// TwinCAT 3 PLC project RS485_Hausbus_LIB
// Title: RS485_Hausbus_Kernal
// Company: NKAutomation
// Author: N.Kersting
// ProjectVersion: 1.5.0.5
// Description: Der reine RS485 Hausbus Kernal.
// ProgramVersion: 3.1.4026.22
// libraries:
//   Tc2_SerialCom, * (Beckhoff Automation GmbH)
//   Tc2_Standard, * (Beckhoff Automation GmbH)
//   Tc2_System, * (Beckhoff Automation GmbH)
//   Tc3_Module, * (Beckhoff Automation GmbH)
// project tree:
//   DUTs/HausBus/BusTaster/ ST_BusTaster6F_Cnt.TcDUT, ST_BusTaster6F_Input.TcDUT, ST_BusTaster6F_Output.TcDUT
//   DUTs/HausBus/CMD/ E_EnumHBCmdRX.TcDUT, E_EnumHBCmdTX.TcDUT, E_EnumHBUnitTX.TcDUT
//   DUTs/HausBus/CYD/ ST_BusCYD6F_Input.TcDUT
//   DUTs/HausBus/Dimmer/ ST_6FDimm.TcDUT, ST_BusDimmer6F_Input.TcDUT, ST_BusDimmer6F_Output.TcDUT
//   DUTs/HausBus/ E_EnumHBDeviceOPMode.TcDUT, E_EnumHBDeviceType.TcDUT, ST_HausBus_Ident.TcDUT
//   DUTs/HausBus/RelaisModul/ ST_16Relais.TcDUT, ST_BusRelais16F_Cnt.TcDUT, ST_BusRelais16F_Input.TcDUT, ST_BusRelais16F_Output.TcDUT
//   DUTs/HausBus/Service/ ST_FiFoMaster_State.TcDUT, ST_RS485ComDeviceStatus.TcDUT, ST_RS485Startup_State.TcDUT
//   DUTs/HausBus/TempSensor/ ST_BusTempSensor4F_Input.TcDUT, ST_BusTempSensor4F_Output.TcDUT
//   GVLs/RS485_HausBus/ GVL_HausBus_ASCII_CONSTANT.TcGVL, GVL_HausBus_CONSTANT.TcGVL, GVL_HausBus_Functions.TcGVL, GVL_HausBus_States.TcGVL, GVL_Times.TcGVL
//   / PlcTask.TcTTO
//   POUs/Hilfsbausteine/ fb_timeDiffLite_libversion.TcPOU
//   POUs/ MAIN.TcPOU
//   POUs/RS485_Hausbus_FB/00_CMD/ fb_RS485HB_StringBuilder.TcPOU, F_RS485HB_TO_ASCII.TcPOU, F_RS485HB_TO_ASCII_RX.TcPOU, F_RS485HB_TO_ASCII_RX_PING.TcPOU
//   POUs/RS485_Hausbus_FB/00_Events/ fb_BusBrsEvent.TcPOU, fb_BusDimmEvent.TcPOU, fb_BusPingEvent.TcPOU (not stored), fb_BusRhdEvent.TcPOU, fb_BusTasterAdvancedEvent_4F.TcPOU, fb_BusTasterAdvancedEvent_6F.TcPOU, fb_BusTasterAdvancedEvent_8F.TcPOU, fb_BusTempEvent.TcPOU
//   POUs/RS485_Hausbus_FB/00_RS485 COM/FB/ fb_FilterArray.TcPOU
//   POUs/RS485_Hausbus_FB/00_RS485 COM/ fb_RS485IdScan.TcPOU
//   POUs/RS485_Hausbus_FB/00_RS485 COM/OLD/ fb_RS485Ping.TcPOU
//   POUs/RS485_Hausbus_FB/00_RS485 COM/RS485_Master/ fb_RS485FiFoMaster.TcPOU, fb_RS485Logger.TcPOU, fb_RS485Startup.TcPOU
//   POUs/RS485_Hausbus_FB/01_BusTaster/ fb_TasterBus6F.TcPOU
//   POUs/RS485_Hausbus_FB/01_CYD/ fb_BusTasterEvent.TcPOU, fb_CYDBus6F.TcPOU, fb_StringConvCYDService.TcPOU, fb_StringConvCYDWeb.TcPOU, fb_StringConvCYDWifi.TcPOU, fb_StringConvTB6F.TcPOU
//   POUs/RS485_Hausbus_FB/01_Dimmer/ fb_DimmerBus6F.TcPOU
//   POUs/RS485_Hausbus_FB/01_RelaisModul/ fb_RelaisBus16F.TcPOU
//   POUs/RS485_Hausbus_FB/01_TempSensor/ fb_TempBus4F.TcPOU
//   POUs/RS485_Hausbus_FB/02_UniBaustein/ fb_RS485PingCheck.TcPOU, fb_UniHBComOperator.TcPOU
//   Project Information/ F_GetCompany.TcPOU, F_GetTitle.TcPOU, F_GetVersion.TcPOU
//   Version/ Global_Version.TcGVL

CONFIGURATION RS485_Hausbus_LIB
    RESOURCE PLC ON TwinCAT3
        TASK PlcTask(INTERVAL := T#10ms, PRIORITY := 20);
        PROGRAM MAIN WITH PlcTask : MAIN;
    END_RESOURCE
END_CONFIGURATION

// ---- DUTs/HausBus/BusTaster/ST_BusTaster6F_Cnt.TcDUT
TYPE ST_BusTaster6F_Cnt :
STRUCT
	dwCntButtons    :ARRAY[1..6] OF DWORD;
END_STRUCT
END_TYPE

// ---- DUTs/HausBus/BusTaster/ST_BusTaster6F_Input.TcDUT
TYPE ST_BusTaster6F_Input :
STRUCT
	diID		:DINT;							(* Device ID ( Steht auf dem Aufkleber und wird zur Identifizierung im BUS benötigt)*)
	sName		:STRING;						(* Name des Tasters (zb- Wohnzimmer1 *)
	iLED      	:ARRAY[1..6] OF INT;     	  	(* gewünschter LED-Zustand (TRUE = 100 %)*)
	iLEDExt    	:ARRAY[1..6] OF INT;     	  	(* gewünschter LED-Zustand (TRUE = 100 %)*)
	iLEDBg		:INT;							(* gewünschte Hintergrundbeleuchtung *)
	bReset		:BOOL;							(* Reset des Tasters (Hardware) *)
	bExecute	:BOOL;							(* Aktivierung des Tasters *)
	bExtOutLED	:BOOL;							(* Verwendet die  Extra Ausgänge für LEDs / Mehr Busaulastung!  *)
	bExtInputs	:BOOL := FALSE;					(* Aktiviert die Externen Inputs *)
END_STRUCT
END_TYPE

// ---- DUTs/HausBus/BusTaster/ST_BusTaster6F_Output.TcDUT
TYPE ST_BusTaster6F_Output :
STRUCT
	bButtons    :ARRAY[1..6] OF BOOL;       (*aktueller Tasterstatus (TRUE = gedrückt)*)
	bButtonsExt :ARRAY[1..6] OF BOOL;       (*aktueller Tasterstatus (TRUE = gedrückt)*)
	
	lrTemp		:LREAL;						(* Temperatur Sensor	*)
	lrRhd		:LREAL;						(* Luftfeuchtigkeit Sensor	*)
	lrBrs		:LREAL;						(* Helligkeit Sensor *)
	
	bCOM			:BOOL;					(*Zeigt die Kommunikation an *)
	bStartupDone	:BOOL;
	
	iState			:BOOL;
	sState			:STRING;
	bError			:BOOL;
	
	tLastUpdateTemp	:TIME;					(* Zeit- Letztes Update Temperatur *)
	tLastUpdateRhd	:TIME;					(* Zeit- Letztes Update Luftfeuchte *)
	tLastUpdateBrs	:TIME;					(* Zeit- Letztes Update Helligkeit *)
	
	sLastUpdateTemp	:STRING(12);			(* Zeit- Letztes Update Temperatur Uhrzeit *)
	sLastUpdateRhd	:STRING(12);			(* Zeit- Letztes Update Luftfeuchte Uhrzeit*)
	sLastUpdateBrs	:STRING(12);			(* Zeit- Letztes Update Helligkeit Uhrzeit*)
	
	dwChanges		:DWORD;					(* Änderungszähler für Startups *)
END_STRUCT
END_TYPE

// ---- DUTs/HausBus/CMD/E_EnumHBCmdRX.TcDUT
{attribute 'qualified_only'}
{attribute 'strict'}
{attribute 'to_string'}
TYPE E_EnumHBCmdRX :
(	
	E_HB_CMD_STATUS := 0,		(* STATUS*)
	E_HB_CMD_rSTATUS := 10,		(* rSTATUS*)
	E_HB_CMD_rCONFIG := 11		(* rCONFIG*)
);
END_TYPE

// ---- DUTs/HausBus/CMD/E_EnumHBCmdTX.TcDUT
{attribute 'qualified_only'}
{attribute 'strict'}
{attribute 'to_string'}
TYPE E_EnumHBCmdTX :
(	
	E_HB_CMD_RESET := 0,	(* RESET*)
	E_HB_CMD_gSTATUS := 100,	(* gSTATUS*)
	E_HB_CMD_gCONFIG := 101,	(* gCONFIG*)
	E_HB_CMD_SET_CFG := 200,	(* SET_CFG*)
	E_HB_CMD_ON := 201,	(* ON*)
	E_HB_CMD_OFF := 202,	(* OFF*)
	E_HB_CMD_SET_MBR := 203,	(* SET_MBR*)
	E_HB_CMD_ON_NP := 204,	(* ON _OHNE Parameter *)
	E_HB_CMD_ON_OFF := 205	(* ON _OFF_ nur über Parameter *)
);
END_TYPE

// ---- DUTs/HausBus/CMD/E_EnumHBUnitTX.TcDUT
{attribute 'qualified_only'}
{attribute 'strict'}
{attribute 'to_string'}
TYPE E_EnumHBUnitTX :
(	
	E_HB_UNIT_SYS := 0,		(* SYS*)
	E_HB_UNIT_BTN := 10,	(* BTN*)
	E_HB_UNIT_OUT := 11,	(* OUT*)
	E_HB_UNIT_LED := 12,	(* LED*)
	E_HB_UNIT_TMP := 13,	(* TMP*)
	E_HB_UNIT_RHD := 14,	(* RHD*)
	E_HB_UNIT_BRS := 15,	(* BRS*)
	E_HB_UNIT_DIM := 16,	(* DIM*)
	E_HB_UNIT_LBN := 17		(* LBN*)
);
END_TYPE

// ---- DUTs/HausBus/CYD/ST_BusCYD6F_Input.TcDUT
TYPE ST_BusCYD6F_Input :
STRUCT
	diID			:DINT;							(* Device ID ( Steht auf dem Aufkleber und wird zur Identifizierung im BUS benötigt)*)
	sName			:STRING;						(* Name des Tasters (zb- Wohnzimmer1 *)
	iLED      		:ARRAY[1..6] OF INT;     	  	(* gewünschter LED-Zustand (TRUE = 100 %)*)
	iLEDExt   	 	:ARRAY[1..6] OF INT;     	  	(* gewünschter LED-Zustand (TRUE = 100 %)*)
	iLEDBg			:INT;							(* gewünschte Hintergrundbeleuchtung *)
	
	
	bReset			:BOOL;							(* Reset des Tasters (Hardware) *)
	bExecute		:BOOL;							(* Aktivierung des Tasters *)
	bExtOutLED		:BOOL;							(* Verwendet die  Extra Ausgänge für LEDs / Mehr Busaulastung!  *)
	
	bServiceMode	:BOOL;
	bService		:BOOL;
	bWifi			:BOOL;
	bWebServer		:BOOL;
END_STRUCT
END_TYPE

// ---- DUTs/HausBus/Dimmer/ST_6FDimm.TcDUT
TYPE ST_6FDimm :
STRUCT
	sLocation			:STRING(28);	
	iDimm	 : ARRAY[1..6] OF INT;
END_STRUCT
END_TYPE

// ---- DUTs/HausBus/Dimmer/ST_BusDimmer6F_Input.TcDUT
TYPE ST_BusDimmer6F_Input :
STRUCT
	diID		:DINT;							(* Device ID ( Steht auf dem Aufkleber und wird zur Identifizierung im BUS benötigt)*)
	sName		:STRING;						(* Name des Tasters (zb- Wohnzimmer1 *)
	iLED      	:ARRAY[1..6] OF INT;     	  	(* gewünschter LED-Zustand (TRUE = 100 %)*)
	iDimmspeed	:INT :=10;						(* Dimmerrampe für alle Kanäle  *)
	bWriteCfg	:BOOL := FALSE;					(* Config write ausführen  *)
	bReset		:BOOL;							(* Reset des Tasters (Hardware) *)
	bExecute	:BOOL;							(* Aktivierung des Tasters *)
	bExtInputs	:BOOL := FALSE;					(* Aktiviert die Externen Inputs *)
END_STRUCT
END_TYPE

// ---- DUTs/HausBus/Dimmer/ST_BusDimmer6F_Output.TcDUT
TYPE ST_BusDimmer6F_Output :
STRUCT
	bInputs		    :ARRAY[1..4] OF BOOL;       (*aktueller Input Status (TRUE = gedrückt)*)
	bCOM			:BOOL;						(*Zeigt die Kommunikation an *)
	bStartupDone	:BOOL;
	
	iState			:BOOL;
	sState			:STRING;
	bError			:BOOL;
	dwChanges		:DWORD;					(* Änderungszähler für Startups *)
END_STRUCT
END_TYPE

// ---- DUTs/HausBus/E_EnumHBDeviceOPMode.TcDUT

TYPE E_EnumHBDeviceOPMode :
(
	E_HB_Device_Init,
	E_HB_Device_CheckID,
	E_HB_Device_EventStartup,
	E_HB_Device_Reset,
	E_HB_Device_WaitCom,
	E_HB_Device_Startup,
	E_HB_Device_OP
);
END_TYPE

// ---- DUTs/HausBus/E_EnumHBDeviceType.TcDUT
TYPE E_EnumHBDeviceType :
(
	E_HB_Device_NV ,
	E_HB_Device_6FTaster,
	E_HB_Device_16FRelais,
	E_HB_Device_6FDimmer,
	E_HB_Device_CYD_1
	
);
END_TYPE

// ---- DUTs/HausBus/RelaisModul/ST_16Relais.TcDUT
TYPE ST_16Relais :
STRUCT
	sLocation			:STRING(28);	
	bOut	 : ARRAY[1..16] OF BOOL;
END_STRUCT
END_TYPE

// ---- DUTs/HausBus/RelaisModul/ST_BusRelais16F_Cnt.TcDUT
TYPE ST_BusRelais16F_Cnt :
STRUCT
	dwCntRelais    :ARRAY[1..16] OF DWORD;
END_STRUCT
END_TYPE

// ---- DUTs/HausBus/RelaisModul/ST_BusRelais16F_Input.TcDUT
TYPE ST_BusRelais16F_Input :
STRUCT
	diID		:DINT;							(* Device ID ( Steht auf dem Aufkleber und wird zur Identifizierung im BUS benötigt)*)
	sName		:STRING;						(* Name des Tasters (zb- Wohnzimmer1 *)
	bOut     	:ARRAY[1..16] OF BOOL;     	  	(* gewünschter Zustand (TRUE = An%)*)
	bReset		:BOOL;							(* Reset des Tasters (Hardware) *)
	bExecute	:BOOL;							(* Aktivierung des Tasters *)
	bExtInputs	:BOOL := FALSE;					(* Aktiviert die Externen Inputs *)
END_STRUCT
END_TYPE

// ---- DUTs/HausBus/RelaisModul/ST_BusRelais16F_Output.TcDUT
TYPE ST_BusRelais16F_Output :
STRUCT
	bInputs		    :ARRAY[1..8] OF BOOL;       (*aktueller Tasterstatus (TRUE = gedrückt)*)
	bCOM			:BOOL;					(*Zeigt die Kommunikation an *)
	bStartupDone	:BOOL;
	
	iState			:BOOL;
	sState			:STRING;
	bError			:BOOL;
	dwChanges		:DWORD;					(* Änderungszähler für Startups *)
END_STRUCT
END_TYPE

// ---- DUTs/HausBus/Service/ST_FiFoMaster_State.TcDUT
TYPE ST_FiFoMaster_State :
STRUCT
	sReceiveString			:STRING(255);		
	lrBusAuslastung			:LREAL;
	bBusy					:BOOL;
	bDone					:BOOL;
	bError					:BOOL;
	iFiFoCount				:INT;
	iFiFoRow				:INT;
	sSendString				:STRING(255);
	sState					:STRING;
	
END_STRUCT
END_TYPE

// ---- DUTs/HausBus/Service/ST_RS485ComDeviceStatus.TcDUT
TYPE ST_RS485ComDeviceStatus :
STRUCT
	diID			:DINT;			
	sState			:STRING;
	bCOM			:BOOL;					(*Zeigt die Kommunikation an *)
	bStartupDone	:BOOL;
	bError			:BOOL;
	
	(* Vorbehalt für Taster *)
	lrTemp			:LREAL;						(* Temperatur Sensor	*)
	lrRhd			:LREAL;						(* Luftfeuchtigkeit Sensor	*)
	lrBrs			:LREAL;						(* Helligkeit Sensor *)
		
	dwChanges		:DWORD;				
END_STRUCT
END_TYPE

// ---- DUTs/HausBus/Service/ST_RS485Startup_State.TcDUT
TYPE ST_RS485Startup_State :
STRUCT
	bBusOk					:BOOL;
	bStartupError			:BOOL;
	sStartupState			:STRING;
	bStartupDone			:BOOL;
END_STRUCT
END_TYPE

// ---- DUTs/HausBus/ST_HausBus_Ident.TcDUT
TYPE ST_HausBus_Ident :
STRUCT
	diID			:DINT;							(* Device ID ( Steht auf dem Aufkleber und wird zur Identifizierung im BUS benötigt)*)
	sName			:STRING;						(* Name des Tasters (zb- Wohnzimmer1 *)	
	sPingIdent		:STRING :='TMP.1.gSTATUS'; 		(* Ping Identifiaktions String, wird bim Pingen gesendet  (Bei Taster = TMP.1.gSTATUS / Relais = OUT.210.rSTATUS / CYD= noch nicht definiert*)
	bUseExtInputs	:BOOL := FALSE;					(* Aktiviert die Externen Inputs *)
END_STRUCT
END_TYPE

// ---- DUTs/HausBus/TempSensor/ST_BusTempSensor4F_Input.TcDUT
TYPE ST_BusTempSensor4F_Input :
STRUCT
	diID		:DINT;							(* Device ID ( Steht auf dem Aufkleber und wird zur Identifizierung im BUS benötigt)*)
	sName		:STRING;						(* Name des Tasters (zb- Wohnzimmer1 *)
	bReset		:BOOL;							(* Reset des ESP32 (Hardware) *)
	bExecute	:BOOL;							(* Aktivierung des Sensors *)
	
	iAnzTempSens :INT := 4;						(* Anzahl der Tempsensoren *)
	bExtInputs	:BOOL := FALSE;					(* Aktiviert die Externen Inputs *)
	
	bWifi			:BOOL;
END_STRUCT
END_TYPE

// ---- DUTs/HausBus/TempSensor/ST_BusTempSensor4F_Output.TcDUT
TYPE ST_BusTempSensor4F_Output :
STRUCT	
	lrTemp			:ARRAY[1..4] OF LREAL;					(* Temperatur Sensor	*)
	
	bCOM			:BOOL;					(*Zeigt die Kommunikation an *)
	bStartupDone	:BOOL;
	
	iState			:BOOL;
	sState			:STRING;
	bError			:BOOL;
	
	tLastUpdateTemp	:ARRAY[1..4] OF TIME;					(* Zeit- Letztes Update Temperatur *)
	
	sLastUpdateTemp	:ARRAY[1..4] OF STRING(12);			(* Zeit- Letztes Update Temperatur Uhrzeit *)
	
	dwChanges		:DWORD;					(* Änderungszähler für Startups *)
END_STRUCT
END_TYPE

// ---- GVLs/RS485_HausBus/GVL_HausBus_ASCII_CONSTANT.TcGVL
{attribute 'qualified_only'}
VAR_GLOBAL CONSTANT
(*==================================================================*)
(* Bibliothek aller ASCII Befehle für alle HAUS-BUS Komponenten *)
(*==================================================================*)

HB_UNIT_SYS : STRING(3) := 'SYS';	(* <SYS>	System *)
HB_UNIT_BRS : STRING(3) := 'BRS';	(* <BRS>	Helligkeit *)
HB_UNIT_BTN : STRING(3) := 'BTN';	(* <BTN>	Button *)
HB_UNIT_DIM : STRING(3) := 'DIM';	(* <DIM>	Dimmer *)
HB_UNIT_LED : STRING(3) := 'LED';	(* <LED>	LED/ Ausgang Taster *)
HB_UNIT_OUT : STRING(3) := 'OUT';	(* <OUT>	Ausgang z.B. Relaismodule  *)
HB_UNIT_RHD : STRING(3) := 'RHD';	(* <RHD>	Luftfeuchtigkeit  *)
HB_UNIT_TMP : STRING(3) := 'TMP';	(* <TMP>	Temperatur  *)
HB_UNIT_LBN : STRING(3) := 'LBN';	(* <LBN>	Hintergrundbeleuchtung (Von Taster) *)

HB_CMD_RESET 	: STRING(7) := 'RESET';		(* <RESET>		Reset des Devices anfordern *)
HB_CMD_gCONFIG 	: STRING(7) := 'gCONFIG';	(* <gCONFIG> 	Config abfragen *)
HB_CMD_gSTATUS 	: STRING(7) := 'gSTATUS';	(* <gSTATUS> 	STATUS abfragen *)
HB_CMD_OFF	 	: STRING(7) := 'OFF';		(* <OFF>		Off Befehl mit Steuerung über Parameter *)
HB_CMD_ON	 	: STRING(7) := 'ON';		(* <ON>			ON Befehl mit Steuerung über Parameter *)
HB_CMD_SET_CFG 	: STRING(7) := 'SET_CFG';	(* <SET_CFG>	Setze Config  *)
HB_CMD_SET_MBR 	: STRING(7) := 'SET_MBR';	(* <SET_MBR>	Setze Hintergrundhelligkeit *)
HB_CMD_ON_NP 	: STRING(7) := 'ON';		(* <ON>			SONDERFUNKTION! Besitzt keine Parameter!  *)
HB_CMD_ON_OFF 	: STRING(7) := '';			(* <ON>			SONDERFUNKTION! Wird über den Parametereingang gesteuert! Wenn P=1 dann 'ON'  wenn P=2 dann 'OFF' *)

HB_RX_rCONFIG	: STRING(7) := 'rCONFIG';	(* <rCONFIG>	Empfang von Config *)
HB_RX_STATUS	: STRING(7) := 'STATUS';	(* <STATUS>		Empfang von Statusnachricht *)
HB_RX_rSTATUS	: STRING(7) := 'rSTATUS';	(* <rSTATUS>	Empfang von Statusantwort *)
END_VAR

// ---- GVLs/RS485_HausBus/GVL_HausBus_CONSTANT.TcGVL
{attribute 'Tc2GvlVarNames'}
VAR_GLOBAL CONSTANT
	(*FiFo*)
	cMaxRowCMDFiFo			:INT := 50; (* Anzahl Maximal mögliche FiFo Zeilen *)
	cMaxScanIDs				:INT := 50;
END_VAR

// ---- GVLs/RS485_HausBus/GVL_HausBus_Functions.TcGVL
{attribute 'Tc2GvlVarNames'}
VAR_GLOBAL
(*================================================================================================================================*)		
(* Changecounter aller Teilnehmer zurücksetzen *)		
(*================================================================================================================================*)	
	bResetChangesCounter_All			:BOOL := FALSE;
END_VAR

// ---- GVLs/RS485_HausBus/GVL_HausBus_States.TcGVL
{attribute 'Tc2GvlVarNames'}
VAR_GLOBAL
	bGlobalPingActive	:BOOL;
END_VAR

// ---- GVLs/RS485_HausBus/GVL_Times.TcGVL
{attribute 'Tc2GvlVarNames'}
VAR_GLOBAL
	
	sGlobClock_SMH					:STRING(12);
END_VAR

// ---- Version/Global_Version.TcGVL
{attribute 'TcGenerated'}
{attribute 'no-analysis'}
{attribute 'linkalways'}
// This function has been automatically generated from the project information.
VAR_GLOBAL CONSTANT
	{attribute 'const_non_replaced'}
	stLibVersion_RS485_Hausbus_Kernal : ST_LibVersion := (iMajor := 1, iMinor := 5, iBuild := 0, iRevision := 5, nFlags := 1, sVersion := '1.5.0.5');
END_VAR

// ---- POUs/MAIN.TcPOU
PROGRAM MAIN
VAR
END_VAR

END_PROGRAM

// ---- POUs/Hilfsbausteine/fb_timeDiffLite_libversion.TcPOU
(*======================================================================================================================================*)
(*fb_timeDiffLite:	Neuer einfacherer Baustein, welcher nur über Start funktioniert *)
(*
Date          	| Version    	| created under        	| Author          	| Remark *)
(*======================================================================================================================================*)
(*03/09/2025   	| 1.00      	| TC3		  			| N.Kersting       | first release *)
(*======================================================================================================================================*)
FUNCTION_BLOCK fb_timeDiffLite_libversion
VAR_INPUT
	I_bStart	:BOOL;
	I_bReset	:BOOL;
END_VAR
VAR_OUTPUT
	Q_tDiffTime	:TIME;
END_VAR
VAR
	tStart	:TIME;
	tStop	:TIME;

	rTrigStart:	R_TRIG;
	rTrigStop:	R_TRIG;
	bMem: BOOL;
END_VAR

rTrigStart(CLK:=I_bStart);

IF	I_bReset	
THEN	
	bMem := FALSE;
	tStart:= T#0S;
	tStop:=T#0S;
ELSE
	
	IF	rTrigStart.Q	
		AND bMem
	THEN	
		bMem := FALSE; 
		tStart:= TIME();
		Q_tDiffTime:=	tStart-tStop;
	END_IF

	IF	rTrigStart.Q
		AND NOT bMem	
	THEN	
		bMem := TRUE;
		tStop:=	TIME();
	END_IF
END_IF

END_FUNCTION_BLOCK

// ---- POUs/RS485_Hausbus_FB/00_CMD/fb_RS485HB_StringBuilder.TcPOU
(*======================================================================================================================================*)
(*//=============================================================================\\
||  _   _ _  __  _         _                        _   _                      ||
|| | \ | | |/ / / \  _   _| |_ ___  _ __ ___   __ _| |_(_) ___  _ __         ||
|| |  \| | ' / / _ \| | | | __/ _ \| '_ ` _ \ / _` | __| |/ _ \| '_ \        ||
|| | |\  | . \/ ___ \ |_| | || (_) | | | | | | (_| | |_| | (_) | | | |       ||
|| |_| \_|_|\_\_/  \_\__,_|\__\___/|_| |_| |_|\__,_|\__|_|\___/|_| |_|       ||
||                                                                             ||
\\=============================================================================//
fb_RS485HB_StringBuilder:	Funktionsbaustein zum zusammenbauen komplexer Strings für Hausbus RS485 Ascii Telegramme		*)
(*
Date          	| Version    	| created under        	| Author          	| Remark *)
(*====================================================================================================================================================*)
(*22/01/2026   	| 1.00      	| TC3		  			| N.Kersting        | first release *)
(*22/01/2026   	| 1.01      	| TC3		  			| N.Kersting        | Erweiterung Array auf 8 Index *)
(*====================================================================================================================================================*)
FUNCTION_BLOCK fb_RS485HB_StringBuilder
VAR_INPUT
	I_bExecute			:BOOL := FALSE;
	I_diID				:DINT;				(* Device ID ( Steht auf dem Aufkleber und wird zur Identifizierung im BUS benötigt)*)
	I_iInstID			:INT;				(* Instanz ID *)
	I_EnumHBUnitTX		:E_EnumHBUnitTX;	(* Unit *)
	I_EnumHBCmdTX		:E_EnumHBCmdTX;		(* Command *)
	I_iCnt				:INT;				(* Anzahl der zusammengefügten Befehle *)
	I_iP1				:ARRAY[1..8] OF INT;				(* Parameter 1 *)
	I_iP2				:ARRAY[1..8] OF INT;				(* Parameter 2 *)
	I_iP3				:ARRAY[1..8] OF INT;				(* Parameter 3 *)
	I_iP4				:ARRAY[1..8] OF INT;				(* Parameter 4 *)
END_VAR
VAR_OUTPUT	
	Q_sOut				:STRING(255);							(* Fertiger Ausgabestring*)	
	Q_bDone				:BOOL;
	Q_bError			:BOOL;
END_VAR
VAR
	IDX 				:INT;
	Trig				:r_trig;
	nLength				:INT;
END_VAR

Trig(CLK:=I_bExecute);

IF Trig.Q
	AND I_bExecute
THEN
	IF I_diID <> 0
	THEN
		IF I_iInstID <> 0
		THEN
			IF I_iCnt <>0
				AND I_iCnt <=8
			THEN
				Q_bError := FALSE;
				
				CASE I_iCnt OF
				(*===========================*)
				0: 	IDX := 0;
					Q_sOut :='';
					
					Q_bDone := TRUE;
					RETURN;
					
				(*===========================*)
				1: 	IDX := 1;
					Q_sOut 	:=		F_RS485HB_TO_ASCII(I_diID,I_iInstID,I_EnumHBUnitTX,I_EnumHBCmdTX,I_iP1[IDX],I_iP2[IDX],I_iP3[IDX],I_iP4[IDX]);
					
					Q_bDone := TRUE;
					
				(*===========================*)
				2: 	IDX := 1;
					Q_sOut 	:=		F_RS485HB_TO_ASCII(I_diID,I_iInstID,I_EnumHBUnitTX,I_EnumHBCmdTX,I_iP1[IDX],I_iP2[IDX],I_iP3[IDX],I_iP4[IDX]);
					IDX := 2;
					Q_sOut 	:=		CONCAT(Q_sOut,F_RS485HB_TO_ASCII(I_diID,I_iInstID+IDX-1,I_EnumHBUnitTX,I_EnumHBCmdTX,I_iP1[IDX],I_iP2[IDX],I_iP3[IDX],I_iP4[IDX]));
					
					Q_bDone := TRUE;
					
				(*===========================*)
				3: 	IDX := 1;
					Q_sOut 	:=		F_RS485HB_TO_ASCII(I_diID,I_iInstID,I_EnumHBUnitTX,I_EnumHBCmdTX,I_iP1[IDX],I_iP2[IDX],I_iP3[IDX],I_iP4[IDX]);
					IDX := 2;
					Q_sOut 	:=		CONCAT(Q_sOut,F_RS485HB_TO_ASCII(I_diID,I_iInstID+IDX-1,I_EnumHBUnitTX,I_EnumHBCmdTX,I_iP1[IDX],I_iP2[IDX],I_iP3[IDX],I_iP4[IDX]));
					IDX := 3;
					Q_sOut 	:=		CONCAT(Q_sOut,F_RS485HB_TO_ASCII(I_diID,I_iInstID+IDX-1,I_EnumHBUnitTX,I_EnumHBCmdTX,I_iP1[IDX],I_iP2[IDX],I_iP3[IDX],I_iP4[IDX]));
					
					Q_bDone := TRUE;
					
				(*===========================*)
				4: 	IDX := 1;
					Q_sOut 	:=		F_RS485HB_TO_ASCII(I_diID,I_iInstID,I_EnumHBUnitTX,I_EnumHBCmdTX,I_iP1[IDX],I_iP2[IDX],I_iP3[IDX],I_iP4[IDX]);
					IDX := 2;
					Q_sOut 	:=		CONCAT(Q_sOut,F_RS485HB_TO_ASCII(I_diID,I_iInstID+IDX-1,I_EnumHBUnitTX,I_EnumHBCmdTX,I_iP1[IDX],I_iP2[IDX],I_iP3[IDX],I_iP4[IDX]));
					IDX := 3;
					Q_sOut 	:=		CONCAT(Q_sOut,F_RS485HB_TO_ASCII(I_diID,I_iInstID+IDX-1,I_EnumHBUnitTX,I_EnumHBCmdTX,I_iP1[IDX],I_iP2[IDX],I_iP3[IDX],I_iP4[IDX]));
					IDX := 4;
					Q_sOut 	:=		CONCAT(Q_sOut,F_RS485HB_TO_ASCII(I_diID,I_iInstID+IDX-1,I_EnumHBUnitTX,I_EnumHBCmdTX,I_iP1[IDX],I_iP2[IDX],I_iP3[IDX],I_iP4[IDX]));
					
					Q_bDone := TRUE;
					
				(*===========================*)
				5: 	IDX := 1;
					Q_sOut 	:=		F_RS485HB_TO_ASCII(I_diID,I_iInstID,I_EnumHBUnitTX,I_EnumHBCmdTX,I_iP1[IDX],I_iP2[IDX],I_iP3[IDX],I_iP4[IDX]);
					IDX := 2;
					Q_sOut 	:=		CONCAT(Q_sOut,F_RS485HB_TO_ASCII(I_diID,I_iInstID+IDX-1,I_EnumHBUnitTX,I_EnumHBCmdTX,I_iP1[IDX],I_iP2[IDX],I_iP3[IDX],I_iP4[IDX]));
					IDX := 3;
					Q_sOut 	:=		CONCAT(Q_sOut,F_RS485HB_TO_ASCII(I_diID,I_iInstID+IDX-1,I_EnumHBUnitTX,I_EnumHBCmdTX,I_iP1[IDX],I_iP2[IDX],I_iP3[IDX],I_iP4[IDX]));
					IDX := 4;
					Q_sOut 	:=		CONCAT(Q_sOut,F_RS485HB_TO_ASCII(I_diID,I_iInstID+IDX-1,I_EnumHBUnitTX,I_EnumHBCmdTX,I_iP1[IDX],I_iP2[IDX],I_iP3[IDX],I_iP4[IDX]));
					IDX := 5;
					Q_sOut 	:=		CONCAT(Q_sOut,F_RS485HB_TO_ASCII(I_diID,I_iInstID+IDX-1,I_EnumHBUnitTX,I_EnumHBCmdTX,I_iP1[IDX],I_iP2[IDX],I_iP3[IDX],I_iP4[IDX]));
					
					Q_bDone := TRUE;
					
				(*===========================*)
				6: 	IDX := 1;
					Q_sOut 	:=		F_RS485HB_TO_ASCII(I_diID,I_iInstID,I_EnumHBUnitTX,I_EnumHBCmdTX,I_iP1[IDX],I_iP2[IDX],I_iP3[IDX],I_iP4[IDX]);
					IDX := 2;
					Q_sOut 	:=		CONCAT(Q_sOut,F_RS485HB_TO_ASCII(I_diID,I_iInstID+IDX-1,I_EnumHBUnitTX,I_EnumHBCmdTX,I_iP1[IDX],I_iP2[IDX],I_iP3[IDX],I_iP4[IDX]));
					IDX := 3;
					Q_sOut 	:=		CONCAT(Q_sOut,F_RS485HB_TO_ASCII(I_diID,I_iInstID+IDX-1,I_EnumHBUnitTX,I_EnumHBCmdTX,I_iP1[IDX],I_iP2[IDX],I_iP3[IDX],I_iP4[IDX]));
					IDX := 4;
					Q_sOut 	:=		CONCAT(Q_sOut,F_RS485HB_TO_ASCII(I_diID,I_iInstID+IDX-1,I_EnumHBUnitTX,I_EnumHBCmdTX,I_iP1[IDX],I_iP2[IDX],I_iP3[IDX],I_iP4[IDX]));
					IDX := 5;
					Q_sOut 	:=		CONCAT(Q_sOut,F_RS485HB_TO_ASCII(I_diID,I_iInstID+IDX-1,I_EnumHBUnitTX,I_EnumHBCmdTX,I_iP1[IDX],I_iP2[IDX],I_iP3[IDX],I_iP4[IDX]));
					IDX := 6;
					Q_sOut 	:=		CONCAT(Q_sOut,F_RS485HB_TO_ASCII(I_diID,I_iInstID+IDX-1,I_EnumHBUnitTX,I_EnumHBCmdTX,I_iP1[IDX],I_iP2[IDX],I_iP3[IDX],I_iP4[IDX]));
					
					Q_bDone := TRUE;
					
				(*===========================*)
				7: 	IDX := 1;
					Q_sOut 	:=		F_RS485HB_TO_ASCII(I_diID,I_iInstID,I_EnumHBUnitTX,I_EnumHBCmdTX,I_iP1[IDX],I_iP2[IDX],I_iP3[IDX],I_iP4[IDX]);
					IDX := 2;
					Q_sOut 	:=		CONCAT(Q_sOut,F_RS485HB_TO_ASCII(I_diID,I_iInstID+IDX-1,I_EnumHBUnitTX,I_EnumHBCmdTX,I_iP1[IDX],I_iP2[IDX],I_iP3[IDX],I_iP4[IDX]));
					IDX := 3;
					Q_sOut 	:=		CONCAT(Q_sOut,F_RS485HB_TO_ASCII(I_diID,I_iInstID+IDX-1,I_EnumHBUnitTX,I_EnumHBCmdTX,I_iP1[IDX],I_iP2[IDX],I_iP3[IDX],I_iP4[IDX]));
					IDX := 4;
					Q_sOut 	:=		CONCAT(Q_sOut,F_RS485HB_TO_ASCII(I_diID,I_iInstID+IDX-1,I_EnumHBUnitTX,I_EnumHBCmdTX,I_iP1[IDX],I_iP2[IDX],I_iP3[IDX],I_iP4[IDX]));
					IDX := 5;
					Q_sOut 	:=		CONCAT(Q_sOut,F_RS485HB_TO_ASCII(I_diID,I_iInstID+IDX-1,I_EnumHBUnitTX,I_EnumHBCmdTX,I_iP1[IDX],I_iP2[IDX],I_iP3[IDX],I_iP4[IDX]));
					IDX := 6;
					Q_sOut 	:=		CONCAT(Q_sOut,F_RS485HB_TO_ASCII(I_diID,I_iInstID+IDX-1,I_EnumHBUnitTX,I_EnumHBCmdTX,I_iP1[IDX],I_iP2[IDX],I_iP3[IDX],I_iP4[IDX]));
					IDX := 7;
					Q_sOut 	:=		CONCAT(Q_sOut,F_RS485HB_TO_ASCII(I_diID,I_iInstID+IDX-1,I_EnumHBUnitTX,I_EnumHBCmdTX,I_iP1[IDX],I_iP2[IDX],I_iP3[IDX],I_iP4[IDX]));
					
					Q_bDone := TRUE;
				
				(*===========================*)
				8: 	IDX := 1;
					Q_sOut 	:=		F_RS485HB_TO_ASCII(I_diID,I_iInstID,I_EnumHBUnitTX,I_EnumHBCmdTX,I_iP1[IDX],I_iP2[IDX],I_iP3[IDX],I_iP4[IDX]);
					IDX := 2;
					Q_sOut 	:=		CONCAT(Q_sOut,F_RS485HB_TO_ASCII(I_diID,I_iInstID+IDX-1,I_EnumHBUnitTX,I_EnumHBCmdTX,I_iP1[IDX],I_iP2[IDX],I_iP3[IDX],I_iP4[IDX]));
					IDX := 3;
					Q_sOut 	:=		CONCAT(Q_sOut,F_RS485HB_TO_ASCII(I_diID,I_iInstID+IDX-1,I_EnumHBUnitTX,I_EnumHBCmdTX,I_iP1[IDX],I_iP2[IDX],I_iP3[IDX],I_iP4[IDX]));
					IDX := 4;
					Q_sOut 	:=		CONCAT(Q_sOut,F_RS485HB_TO_ASCII(I_diID,I_iInstID+IDX-1,I_EnumHBUnitTX,I_EnumHBCmdTX,I_iP1[IDX],I_iP2[IDX],I_iP3[IDX],I_iP4[IDX]));
					IDX := 5;
					Q_sOut 	:=		CONCAT(Q_sOut,F_RS485HB_TO_ASCII(I_diID,I_iInstID+IDX-1,I_EnumHBUnitTX,I_EnumHBCmdTX,I_iP1[IDX],I_iP2[IDX],I_iP3[IDX],I_iP4[IDX]));
					IDX := 6;
					Q_sOut 	:=		CONCAT(Q_sOut,F_RS485HB_TO_ASCII(I_diID,I_iInstID+IDX-1,I_EnumHBUnitTX,I_EnumHBCmdTX,I_iP1[IDX],I_iP2[IDX],I_iP3[IDX],I_iP4[IDX]));
					IDX := 7;
					Q_sOut 	:=		CONCAT(Q_sOut,F_RS485HB_TO_ASCII(I_diID,I_iInstID+IDX-1,I_EnumHBUnitTX,I_EnumHBCmdTX,I_iP1[IDX],I_iP2[IDX],I_iP3[IDX],I_iP4[IDX]));
					IDX := 8;
					Q_sOut 	:=		CONCAT(Q_sOut,F_RS485HB_TO_ASCII(I_diID,I_iInstID+IDX-1,I_EnumHBUnitTX,I_EnumHBCmdTX,I_iP1[IDX],I_iP2[IDX],I_iP3[IDX],I_iP4[IDX]));
					
					Q_bDone := TRUE;	
				END_CASE
				
				nLength :=	LEN(Q_sOut);
				RETURN;
			ELSE
				Q_bError := TRUE;
			END_IF
		ELSE
			Q_bError := TRUE;
		END_IF
	ELSE
		Q_bError := TRUE;
	END_IF
ELSIF
	NOT I_bExecute
THEN
	Q_bDone := FALSE;
	Q_sOut :='x';
END_IF

END_FUNCTION_BLOCK

// ---- POUs/RS485_Hausbus_FB/00_CMD/F_RS485HB_TO_ASCII.TcPOU
(*======================================================================================================================================*)
(*//=============================================================================\\
||  _   _ _  __  _         _                        _   _                      ||
|| | \ | | |/ / / \  _   _| |_ ___  _ __ ___   __ _| |_(_) ___  _ __         ||
|| |  \| | ' / / _ \| | | | __/ _ \| '_ ` _ \ / _` | __| |/ _ \| '_ \        ||
|| | |\  | . \/ ___ \ |_| | || (_) | | | | | | (_| | |_| | (_) | | | |       ||
|| |_| \_|_|\_\_/  \_\__,_|\__\___/|_| |_| |_|\__,_|\__|_|\___/|_| |_|       ||
||                                                                             ||
\\=============================================================================//
F_RS485HB_TO_ASCII:	Funktion um Hausbus Ascii Strings zu generieren		*)
(*
Date          	| Version    	| created under        	| Author          	| Remark *)
(*====================================================================================================================================================*)
(*22/01/2026   	| 1.00      	| TC3		  			| N.Kersting        | first release *)
(*====================================================================================================================================================*)
FUNCTION F_RS485HB_TO_ASCII : STRING(255)
VAR_INPUT
	I_diID				:DINT;				(* Device ID ( Steht auf dem Aufkleber und wird zur Identifizierung im BUS benötigt)*)
	I_iInstID			:INT;				(* Instanz ID *)
	I_EnumHBUnitTX		:E_EnumHBUnitTX;	(* Unit *)
	I_EnumHBCmdTX		:E_EnumHBCmdTX;		(* Command *)
	I_iP1				:INT;				(* Parameter 1 *)
	I_iP2				:INT;				(* Parameter 2 *)
	I_iP3				:INT;				(* Parameter 3 *)
	I_iP4				:INT;				(* Parameter 4 *)
END_VAR
VAR
	sStartZeichen		:BYTE := 16#FD;				(* Startzeichen Präfix *)
	sEndZeichen			:BYTE := 16#FE;				(* Endzeichen Suffix *)
	
	Q_sOut			:STRING(255);
	sUnit			:STRING(3);
	bInvalidUnit	:BOOL;
	
	sCMD			:STRING(7);
	bInvalidCMD		:BOOL;
	
	iParam			:INT;
END_VAR

bInvalidUnit := FALSE;
bInvalidCMD := FALSE;

CASE I_EnumHBUnitTX OF
E_EnumHBUnitTX.E_HB_UNIT_SYS:  sUnit :=	GVL_HausBus_ASCII_CONSTANT.HB_UNIT_SYS; 	
E_EnumHBUnitTX.E_HB_UNIT_BRS:  sUnit :=	GVL_HausBus_ASCII_CONSTANT.HB_UNIT_BRS; 	
E_EnumHBUnitTX.E_HB_UNIT_BTN:  sUnit :=	GVL_HausBus_ASCII_CONSTANT.HB_UNIT_BTN; 	
E_EnumHBUnitTX.E_HB_UNIT_DIM:  sUnit :=	GVL_HausBus_ASCII_CONSTANT.HB_UNIT_DIM; 	
E_EnumHBUnitTX.E_HB_UNIT_LED:  sUnit :=	GVL_HausBus_ASCII_CONSTANT.HB_UNIT_LED; 	
E_EnumHBUnitTX.E_HB_UNIT_OUT:  sUnit :=	GVL_HausBus_ASCII_CONSTANT.HB_UNIT_OUT; 
E_EnumHBUnitTX.E_HB_UNIT_RHD:  sUnit :=	GVL_HausBus_ASCII_CONSTANT.HB_UNIT_RHD; 
E_EnumHBUnitTX.E_HB_UNIT_TMP:  sUnit :=	GVL_HausBus_ASCII_CONSTANT.HB_UNIT_TMP; 
E_EnumHBUnitTX.E_HB_UNIT_LBN:  sUnit :=	GVL_HausBus_ASCII_CONSTANT.HB_UNIT_LBN; 
ELSE
	bInvalidUnit := TRUE;
	RETURN;
END_CASE

CASE I_EnumHBCmdTX OF
E_EnumHBCmdTX.E_HB_CMD_RESET:		sCMD :=		GVL_HausBus_ASCII_CONSTANT.HB_CMD_RESET;	iParam := 0;
E_EnumHBCmdTX.E_HB_CMD_gCONFIG:		sCMD :=		GVL_HausBus_ASCII_CONSTANT.HB_CMD_gCONFIG;	iParam := 0;
E_EnumHBCmdTX.E_HB_CMD_gSTATUS:		sCMD :=		GVL_HausBus_ASCII_CONSTANT.HB_CMD_gSTATUS;	iParam := 0;
E_EnumHBCmdTX.E_HB_CMD_OFF:			sCMD :=		GVL_HausBus_ASCII_CONSTANT.HB_CMD_OFF;		iParam := 0;
E_EnumHBCmdTX.E_HB_CMD_ON:			sCMD :=		GVL_HausBus_ASCII_CONSTANT.HB_CMD_ON;		iParam := 1;
E_EnumHBCmdTX.E_HB_CMD_SET_CFG:		sCMD :=		GVL_HausBus_ASCII_CONSTANT.HB_CMD_SET_CFG;	iParam := 2;
E_EnumHBCmdTX.E_HB_CMD_SET_MBR:		sCMD :=		GVL_HausBus_ASCII_CONSTANT.HB_CMD_SET_MBR;	iParam := 1;
E_EnumHBCmdTX.E_HB_CMD_ON_NP:		sCMD :=		GVL_HausBus_ASCII_CONSTANT.HB_CMD_ON_NP;	iParam := 0;
E_EnumHBCmdTX.E_HB_CMD_ON_OFF:																iParam := 0;

	(* Spezialbefehl On Off über Parameter *)
	CASE I_iP1 OF
	0: 	sCMD :=		GVL_HausBus_ASCII_CONSTANT.HB_CMD_OFF;
	1: 	sCMD :=		GVL_HausBus_ASCII_CONSTANT.HB_CMD_ON;
	ELSE
		sCMD :=		'';
	END_CASE
ELSE
	bInvalidCMD := TRUE;
	RETURN;
END_CASE

IF I_diID > 0
THEN
	IF I_iInstID > 0
	THEN
		IF NOT bInvalidUnit
			AND NOT bInvalidCMD
		THEN
		
			Q_sOut :=	CONCAT(F_ToCHR(sStartZeichen),DINT_TO_STRING(I_diID));
			Q_sOut :=	CONCAT(Q_sOut,'.');
			Q_sOut :=	CONCAT(Q_sOut,sUnit);
			Q_sOut :=	CONCAT(Q_sOut,'.');
			Q_sOut :=	CONCAT(Q_sOut,INT_TO_STRING(I_iInstID));
			Q_sOut :=	CONCAT(Q_sOut,'.');
			Q_sOut :=	CONCAT(Q_sOut,sCMD);
			
			CASE iParam OF
			0:	Q_sOut :=	CONCAT(Q_sOut,F_ToCHR(sEndZeichen));
			
			1:	Q_sOut :=	CONCAT(Q_sOut,'.');
				Q_sOut :=	CONCAT(Q_sOut,INT_TO_STRING(I_iP1));
				Q_sOut :=	CONCAT(Q_sOut,F_ToCHR(sEndZeichen));
				
			2:	Q_sOut :=	CONCAT(Q_sOut,'.');
				Q_sOut :=	CONCAT(Q_sOut,INT_TO_STRING(I_iP1));
				Q_sOut :=	CONCAT(Q_sOut,'.');
				Q_sOut :=	CONCAT(Q_sOut,INT_TO_STRING(I_iP2));
				Q_sOut :=	CONCAT(Q_sOut,F_ToCHR(sEndZeichen));
				
			3:	Q_sOut :=	CONCAT(Q_sOut,'.');
				Q_sOut :=	CONCAT(Q_sOut,INT_TO_STRING(I_iP1));
				Q_sOut :=	CONCAT(Q_sOut,'.');
				Q_sOut :=	CONCAT(Q_sOut,INT_TO_STRING(I_iP2));
				Q_sOut :=	CONCAT(Q_sOut,'.');
				Q_sOut :=	CONCAT(Q_sOut,INT_TO_STRING(I_iP3));
				Q_sOut :=	CONCAT(Q_sOut,F_ToCHR(sEndZeichen));
				
			4:	Q_sOut :=	CONCAT(Q_sOut,'.');
				Q_sOut :=	CONCAT(Q_sOut,INT_TO_STRING(I_iP1));
				Q_sOut :=	CONCAT(Q_sOut,'.');
				Q_sOut :=	CONCAT(Q_sOut,INT_TO_STRING(I_iP2));
				Q_sOut :=	CONCAT(Q_sOut,'.');
				Q_sOut :=	CONCAT(Q_sOut,INT_TO_STRING(I_iP3));
				Q_sOut :=	CONCAT(Q_sOut,'.');
				Q_sOut :=	CONCAT(Q_sOut,INT_TO_STRING(I_iP4));
				Q_sOut :=	CONCAT(Q_sOut,F_ToCHR(sEndZeichen));
				
			END_CASE
		END_IF
	END_IF
END_IF

F_RS485HB_TO_ASCII:=Q_sOut;
RETURN;

END_FUNCTION

// ---- POUs/RS485_Hausbus_FB/00_CMD/F_RS485HB_TO_ASCII_RX.TcPOU
(*======================================================================================================================================*)
(*//=============================================================================\\
||  _   _ _  __  _         _                        _   _                      ||
|| | \ | | |/ / / \  _   _| |_ ___  _ __ ___   __ _| |_(_) ___  _ __         ||
|| |  \| | ' / / _ \| | | | __/ _ \| '_ ` _ \ / _` | __| |/ _ \| '_ \        ||
|| | |\  | . \/ ___ \ |_| | || (_) | | | | | | (_| | |_| | (_) | | | |       ||
|| |_| \_|_|\_\_/  \_\__,_|\__\___/|_| |_| |_|\__,_|\__|_|\___/|_| |_|       ||
||                                                                             ||
\\=============================================================================//
F_RS485HB_TO_ASCII_RX:	Sonderfunktion um Hausbus Ascii Strings zu generieren speziell für Suchstring		*)
(*
Date          	| Version    	| created under        	| Author          	| Remark *)
(*====================================================================================================================================================*)
(*22/01/2026   	| 1.00      	| TC3		  			| N.Kersting        | first release *)
(*====================================================================================================================================================*)
FUNCTION F_RS485HB_TO_ASCII_RX : STRING(255)
VAR_INPUT
	I_diID				:DINT;				(* Device ID ( Steht auf dem Aufkleber und wird zur Identifizierung im BUS benötigt)*)
	I_iInstID			:INT;				(* Instanz ID *)
	I_EnumHBUnitTX		:E_EnumHBUnitTX;	(* Unit *)
	I_EnumHBCmdRX		:E_EnumHBCmdRX;		(* Command *)
	I_iP1				:INT;				(* Parameter 1 *)
	
END_VAR
VAR
	sStartZeichen		:BYTE := 16#FD;				(* Startzeichen Präfix *)
	sEndZeichen			:BYTE := 16#FE;				(* Endzeichen Suffix *)
	
	Q_sOut			:STRING(255);
	sUnit			:STRING(3);
	bInvalidUnit	:BOOL;
	
	sCMD			:STRING(7);
	bInvalidCMD		:BOOL;
	
	iParam			:INT;
END_VAR

bInvalidUnit := FALSE;
bInvalidCMD := FALSE;

CASE I_EnumHBUnitTX OF
E_EnumHBUnitTX.E_HB_UNIT_SYS:  sUnit :=	GVL_HausBus_ASCII_CONSTANT.HB_UNIT_SYS; 	iParam := 0;	
E_EnumHBUnitTX.E_HB_UNIT_BRS:  sUnit :=	GVL_HausBus_ASCII_CONSTANT.HB_UNIT_BRS; 	iParam := 0;
E_EnumHBUnitTX.E_HB_UNIT_BTN:  sUnit :=	GVL_HausBus_ASCII_CONSTANT.HB_UNIT_BTN; 	iParam := 1;
E_EnumHBUnitTX.E_HB_UNIT_DIM:  sUnit :=	GVL_HausBus_ASCII_CONSTANT.HB_UNIT_DIM; 	iParam := 0;
E_EnumHBUnitTX.E_HB_UNIT_LED:  sUnit :=	GVL_HausBus_ASCII_CONSTANT.HB_UNIT_LED; 	iParam := 0;
E_EnumHBUnitTX.E_HB_UNIT_OUT:  sUnit :=	GVL_HausBus_ASCII_CONSTANT.HB_UNIT_OUT; 	iParam := 1;
E_EnumHBUnitTX.E_HB_UNIT_RHD:  sUnit :=	GVL_HausBus_ASCII_CONSTANT.HB_UNIT_RHD; 	iParam := 0;
E_EnumHBUnitTX.E_HB_UNIT_TMP:  sUnit :=	GVL_HausBus_ASCII_CONSTANT.HB_UNIT_TMP; 	iParam := 0;
E_EnumHBUnitTX.E_HB_UNIT_LBN:  sUnit :=	GVL_HausBus_ASCII_CONSTANT.HB_UNIT_LBN; 	iParam := 0;
ELSE
	bInvalidUnit := TRUE;
	RETURN;
END_CASE

CASE I_EnumHBCmdRX OF
E_EnumHBCmdRX.E_HB_CMD_rCONFIG:		sCMD :=		GVL_HausBus_ASCII_CONSTANT.HB_RX_rCONFIG;	
E_EnumHBCmdRX.E_HB_CMD_rSTATUS:		sCMD :=		GVL_HausBus_ASCII_CONSTANT.HB_RX_rSTATUS;	
E_EnumHBCmdRX.E_HB_CMD_STATUS:		sCMD :=		GVL_HausBus_ASCII_CONSTANT.HB_RX_STATUS;
ELSE
	bInvalidCMD := TRUE;
	RETURN;
END_CASE

IF I_diID > 0
THEN
	IF I_iInstID > 0
	THEN
		IF NOT bInvalidUnit
			AND NOT bInvalidCMD
		THEN
					
			Q_sOut :=	CONCAT(F_ToCHR(sStartZeichen),DINT_TO_STRING(I_diID));
			Q_sOut :=	CONCAT(Q_sOut,'.');
			Q_sOut :=	CONCAT(Q_sOut,sUnit);
			Q_sOut :=	CONCAT(Q_sOut,'.');
			Q_sOut :=	CONCAT(Q_sOut,INT_TO_STRING(I_iInstID));
			Q_sOut :=	CONCAT(Q_sOut,'.');
			Q_sOut :=	CONCAT(Q_sOut,sCMD);
			
			CASE iParam OF
			0:	Q_sOut :=	CONCAT(Q_sOut,'.');
				(*Q_sOut :=	CONCAT(Q_sOut,F_ToCHR(sEndZeichen));*)
			1:	Q_sOut :=	CONCAT(Q_sOut,'.');
				Q_sOut :=	CONCAT(Q_sOut,INT_TO_STRING(I_iP1));
				Q_sOut :=	CONCAT(Q_sOut,F_ToCHR(sEndZeichen));	
			END_CASE
		END_IF
	END_IF
END_IF

F_RS485HB_TO_ASCII_RX:=Q_sOut;
RETURN;

END_FUNCTION

// ---- POUs/RS485_Hausbus_FB/00_CMD/F_RS485HB_TO_ASCII_RX_PING.TcPOU
(*======================================================================================================================================*)
(*//=============================================================================\\
||  _   _ _  __  _         _                        _   _                      ||
|| | \ | | |/ / / \  _   _| |_ ___  _ __ ___   __ _| |_(_) ___  _ __         ||
|| |  \| | ' / / _ \| | | | __/ _ \| '_ ` _ \ / _` | __| |/ _ \| '_ \        ||
|| | |\  | . \/ ___ \ |_| | || (_) | | | | | | (_| | |_| | (_) | | | |       ||
|| |_| \_|_|\_\_/  \_\__,_|\__\___/|_| |_| |_|\__,_|\__|_|\___/|_| |_|       ||
||                                                                             ||
\\=============================================================================//
F_RS485HB_TO_ASCII_RX_PING:	Sonderfunktion um Hausbus Ascii Strings zu generieren speziell für Suchstring		*)
(*
Date          	| Version    	| created under        	| Author          	| Remark *)
(*====================================================================================================================================================*)
(*22/01/2026   	| 1.00      	| TC3		  			| N.Kersting        | first release *)
(*====================================================================================================================================================*)
FUNCTION F_RS485HB_TO_ASCII_RX_PING : STRING(255)
VAR_INPUT
	I_diID				:DINT;				(* Device ID ( Steht auf dem Aufkleber und wird zur Identifizierung im BUS benötigt)*)	
END_VAR
VAR
	sStartZeichen		:BYTE := 16#FD;				(* Startzeichen Präfix *)
	sEndZeichen			:BYTE := 16#FE;				(* Endzeichen Suffix *)
	Q_sOut				:STRING[255);
	
END_VAR


IF I_diID > 0
THEN
	Q_sOut :=	CONCAT(F_ToCHR(sStartZeichen),DINT_TO_STRING(I_diID));
END_IF

F_RS485HB_TO_ASCII_RX_PING:=Q_sOut;
RETURN;

END_FUNCTION

// ---- POUs/RS485_Hausbus_FB/00_Events/fb_BusBrsEvent.TcPOU
(*======================================================================================================================================*)
(*//=============================================================================\\
||  _   _ _  __  _         _                        _   _                      ||
|| | \ | | |/ / / \  _   _| |_ ___  _ __ ___   __ _| |_(_) ___  _ __         ||
|| |  \| | ' / / _ \| | | | __/ _ \| '_ ` _ \ / _` | __| |/ _ \| '_ \        ||
|| | |\  | . \/ ___ \ |_| | || (_) | | | | | | (_| | |_| | (_) | | | |       ||
|| |_| \_|_|\_\_/  \_\__,_|\__\___/|_| |_| |_|\__,_|\__|_|\___/|_| |_|       ||
||                                                                             ||
\\=============================================================================//
fb_BusBrsEvent:				Dieser Baustein sieht Helligkeit Events.  *)
(*
Date          	| Version    	| created under        	| Author          	| Remark *)
(*====================================================================================================================================================*)
(*29/04/2025   	| 1.00      		| TC3		  		| N.Kersting       | first release *)
(*14/08/2025   	| 1.01      		| TC3		  		| N.Kersting       | Startup Schrittkette Implementiert um Effizienter zu werden*)
(*27/08/2025   	| 1.02      		| TC3		  		| N.Kersting       | Reset hinzugefügt / Startup Done Ausgang *)
(*03/09/2025   	| 1.03      		| TC3		  		| N.Kersting       | Wenn der Wert sich erneuert, wird die Zeit gemessen zwischen den Updates *)
(*07/09/2025   	| 1.04      		| TC3		  		| N.Kersting       | Zykluszeit Optimierung, es wird nur gelesen, wenn String gefüllt ist *)
(*09/09/2025   	| 1.05      		| TC3		  		| N.Kersting       | Zykluszeit Optimierung, Wirklich nur einen Zyklus suchen *)
(*25/01/2026   	| 2.00      		| TC3		  		| N.Kersting       | Suchstring umstellung auf ASCII_RS485 Funktion *)
(*====================================================================================================================================================*)
FUNCTION_BLOCK fb_BusBrsEvent
VAR_INPUT
	 I_bExecute				:BOOL := TRUE;	// Aktiviert den Baustein 
	 I_diID        			:DINT;     // Geräte-ID (z.B. '12345')
	 I_iInstID				:INT 	:=	17;
	 I_sReceivedString		:STRING(255);	
	 I_bReset				:BOOL;
END_VAR
VAR_OUTPUT
	Q_lrBrs					:LREAL;
	Q_bStartupDone			:BOOL;
	Q_tUpdate				:TIME;
	Q_sLastUpdate			:STRING(12);
END_VAR
VAR	
	findStringTemp			:STRING(255);	(* Wird für TMP/ BRS/ RHD verwendet *)

	sTemp1					:STRING(255);
	sTemp2					:STRING(255);
	
	startPos : INT;
		
	iFindString	:int;
	icnt					:INT ;
	r_trigCnt				:r_trig;
		
	bStartupStart			:BOOL;
	bStartupDone			:BOOL;
	
	iStartup				:INT;
	fbtimeDiff				:fb_timeDiffLite_libversion;
	bUpdated				: BOOL;
			
	sLastString				:STRING(255);
	bNeedProcess			:BOOL;
END_VAR

r_trigCnt();

(* Automatische Fehlererkennung *)
IF NOT I_bExecute
	OR (I_diID = 0)
	OR (I_iInstID = 0)
THEN
	iStartup := 0;
END_IF

(* Warten, ob der String sich geändert hat*)
bNeedProcess :=	(I_sReceivedString <> sLastString) 
				AND (I_sReceivedString <> '');

CASE iStartup OF 
(*=====================================*)
0 :	(* INIT *)
	bStartupDone := FALSE;
	bStartupStart := FALSE;
	sTemp2 :=sTemp1 := '0';
	r_trigCnt.CLK := FALSE;
	bNeedProcess := FALSE;
	sLastString := '';
	
	IF I_bExecute
		AND NOT bStartupDone
		AND NOT I_bReset
		AND (I_diID <> 0)
		AND (I_iInstID <>0)
	THEN
		bStartupStart := TRUE;
		iStartup := iStartup +10;
	END_IF
	
(*=====================================*)
10 :(* String vorbereiten *)	
	findStringTemp := F_RS485HB_TO_ASCII_RX(
							I_diID			:= I_diID, 
							I_iInstID		:= I_iInstID,	
							I_EnumHBUnitTX	:= E_EnumHBUnitTX.E_HB_UNIT_BRS, 	
							I_EnumHBCmdRX	:= E_EnumHBCmdRX.E_HB_CMD_STATUS , 
							I_iP1			:= 0);
								
	iStartup := 999;
	
(*=====================================*)
999 :(* READY *)
	bStartupDone := TRUE;
	
	IF I_bReset 
	THEN
		iStartup := 0;
	ELSE
		IF bNeedProcess
		THEN
			iFindString :=	FIND(I_sReceivedString,findStringTemp);
			
			IF iFindString>0
			THEN
				r_trigCnt.CLK := TRUE;
				startPos := iFindString; // Position des Suchstrings       
				(*Temperatur steht direkt nach dem Suchstring*)
				startPos := startPos + LEN(findStringTemp); (*Startposition für Temperatur*)
				(* Temperatur bis zum nächsten Komma oder Ende auslesen (maximal 6 Zeichen: z.B. 24,74)*)
				sTemp1 := MID(I_sReceivedString, 5, startPos);
				(*Dezimalpunkt für STRING_TO_LREAL anpassen, falls nötig *)
				sTemp1 := REPLACE(sTemp1, '.',1,3); (* 1. Vorkommen ersetzen *)
			ELSE
				r_trigCnt.CLK := FALSE;
			END_IF
			
			sLastString :=	I_sReceivedString;	(* Letzten String Speichern *)
		END_IF
	END_IF
	
	Q_lrBrs := STRING_TO_LREAL(sTemp1);

	(* Counter für Diagnose *)
	IF r_trigCnt.Q
	THEN
		Q_sLastUpdate :=	sGlobClock_SMH;	(* Globale Uhrzeit SMH*)
		
		bUpdated := TRUE;
		sTemp2 :=	I_sReceivedString;	(* Speichern der Werte *)
		icnt := icnt+1;
	ELSE
		bUpdated := FALSE;
	END_IF
	
END_CASE

Q_bStartupDone := bStartupDone;

(*=====================================*)
(* Zeitmessung zwischen den Updates *)
fbtimeDiff(
	I_bStart:= 			bUpdated, 
	I_bReset:= 			I_bReset, 
	Q_tDiffTime=>		Q_tUpdate);

END_FUNCTION_BLOCK

// ---- POUs/RS485_Hausbus_FB/00_Events/fb_BusDimmEvent.TcPOU
(*======================================================================================================================================*)
(*//=============================================================================\\
||  _   _ _  __  _         _                        _   _                      ||
|| | \ | | |/ / / \  _   _| |_ ___  _ __ ___   __ _| |_(_) ___  _ __         ||
|| |  \| | ' / / _ \| | | | __/ _ \| '_ ` _ \ / _` | __| |/ _ \| '_ \        ||
|| | |\  | . \/ ___ \ |_| | || (_) | | | | | | (_| | |_| | (_) | | | |       ||
|| |_| \_|_|\_\_/  \_\__,_|\__\___/|_| |_| |_|\__,_|\__|_|\___/|_| |_|       ||
||                                                                             ||
\\=============================================================================//
fb_BusDimmEvent:	Dieser Baustein sieht Dimmer Events und wertet diese aus, möglichst effizient.
								  *)
(*
Date          	| Version    	| created under        	| Author          	| Remark *)
(*====================================================================================================================================================*)
(*13/01/2026   	| 1.00      		| TC3		  		| N.Kersting       | first release *)
(*25/01/2026   	| 2.00      		| TC3		  		| N.Kersting       | Suchstring umstellung auf ASCII_RS485 Funktion *)
(*====================================================================================================================================================*)
FUNCTION_BLOCK fb_BusDimmEvent
VAR_INPUT
	 I_bExecute				:BOOL := TRUE;	// Aktiviert den Baustein 
	 I_bReset				:BOOL;
	 I_diID        			:DINT;     // Geräte-ID (z.B. '12345')
	 I_iInstID				:INT 	:=	17;
	 I_sReceivedString		:STRING(255);	
END_VAR
VAR_OUTPUT
	Q_iOut					:ARRAY[1..6] OF  INT;
	Q_bStartupDone			:BOOL;
END_VAR
VAR
	i						:INT;
	findString0				:ARRAY[1..6] OF STRING(255);
	
	iFindString				:ARRAY[1..6] OF INT;
	startPos 				:ARRAY[1..6] OF INT;
	
	bStartupStart			:BOOL;
	bStartupDone			:BOOL;
	
	iStartup				:INT;
	
	sLastString				:STRING(255);
	bNeedProcess			:BOOL;
END_VAR

(* Automatische Fehlererkennung *)
IF NOT I_bExecute
	OR (I_diID = 0)
	OR (I_iInstID = 0)
THEN
	iStartup := 0;
END_IF

(* Warten, ob der String sich geändert hat*)
bNeedProcess :=	(I_sReceivedString <> sLastString) 
				AND (I_sReceivedString <> '');

CASE iStartup OF 
(*=====================================*)
0 :	(* INIT *)
	bStartupDone := FALSE;
	bStartupStart := FALSE;
	bNeedProcess := FALSE;
	sLastString := '';
	
	FOR i := 1 TO 6 BY 1 DO
		
		Q_iOut[i] := 0;
		
	END_FOR	
	
	IF I_bExecute
		AND NOT bStartupDone
		AND NOT I_bReset
		AND (I_diID <> 0)
		AND (I_iInstID <>0)
	THEN
		i := 1;
		bStartupStart := TRUE;
		iStartup := iStartup +10;
	END_IF
	
(*=====================================*)
10 :(* String vorbereiten *)	
		
	FOR i := 1 TO 6 BY 1 DO
		findString0[i] := F_RS485HB_TO_ASCII_RX(
							I_diID			:= I_diID, 
							I_iInstID		:= I_iInstID+i-1,	
							I_EnumHBUnitTX	:= E_EnumHBUnitTX.E_HB_UNIT_DIM, 	
							I_EnumHBCmdRX	:= E_EnumHBCmdRX.E_HB_CMD_rSTATUS , 
							I_iP1			:= 0);
	END_FOR
	
	
	IF i >= 6 THEN
		bStartupStart := FALSE;
		iStartup := 999;
	END_IF
	
(*=====================================*)
999 :(* READY *)
	bStartupDone := TRUE;
	
	IF I_bReset 
	THEN
		iStartup := 0;
	ELSE
		IF bNeedProcess
		THEN
			FOR i := 1 TO 6 BY 1 DO					
				iFindString[i] :=	FIND(I_sReceivedString,findString0[i]);
			
				IF iFindString[i]>0
				THEN
					startPos[i] := iFindString[i]; // Position des Suchstrings       
					(*Dimmer steht direkt nach dem Suchstring*)
					startPos[i] := startPos[i] + LEN(findString0[i]); (*Startposition für Temperatur*)
					(* Dimmer bis zum nächsten Komma oder Ende auslesen (maximal 6 Zeichen: z.B. 100)*)
					Q_iOut[i] := STRING_TO_INT(MID(I_sReceivedString, 3, startPos[i]));
				END_IF
			END_FOR	
			sLastString :=	I_sReceivedString;	(* Letzten String Speichern *)
		END_IF
	END_IF
END_CASE

Q_bStartupDone := bStartupDone;

END_FUNCTION_BLOCK

// ---- POUs/RS485_Hausbus_FB/00_Events/fb_BusRhdEvent.TcPOU
(*======================================================================================================================================*)
(*//=============================================================================\\
||  _   _ _  __  _         _                        _   _                      ||
|| | \ | | |/ / / \  _   _| |_ ___  _ __ ___   __ _| |_(_) ___  _ __         ||
|| |  \| | ' / / _ \| | | | __/ _ \| '_ ` _ \ / _` | __| |/ _ \| '_ \        ||
|| | |\  | . \/ ___ \ |_| | || (_) | | | | | | (_| | |_| | (_) | | | |       ||
|| |_| \_|_|\_\_/  \_\__,_|\__\___/|_| |_| |_|\__,_|\__|_|\___/|_| |_|       ||
||                                                                             ||
\\=============================================================================//
fb_BusRhdEvent:				Dieser Baustein sieht Feuchtigkeit Events.  *)
(*
Date          	| Version    	| created under        	| Author          	| Remark *)
(*====================================================================================================================================================*)
(*29/04/2025   	| 1.00      		| TC3		  		| N.Kersting       | first release *)
(*14/08/2025   	| 1.01      		| TC3		  		| N.Kersting       | Startup Schrittkette Implementiert um Effizienter zu werden*)
(*27/08/2025   	| 1.02      		| TC3		  		| N.Kersting       | Reset hinzugefügt / Startup Done Ausgang *)
(*03/09/2025   	| 1.03      		| TC3		  		| N.Kersting       | Wenn der Wert sich erneuert, wird die Zeit gemessen zwischen den Updates *)
(*07/09/2025   	| 1.04      		| TC3		  		| N.Kersting       | Zykluszeit Optimierung, es wird nur gelesen, wenn String gefüllt ist *)
(*09/09/2025   	| 1.05      		| TC3		  		| N.Kersting       | Zykluszeit Optimierung, Wirklich nur einen Zyklus suchen *)
(*25/01/2026   	| 2.00      		| TC3		  		| N.Kersting       | Suchstring umstellung auf ASCII_RS485 Funktion *)
(*====================================================================================================================================================*)
FUNCTION_BLOCK fb_BusRhdEvent
VAR_INPUT
	 I_bExecute				:BOOL := TRUE;	// Aktiviert den Baustein 
	 I_diID        			:DINT;     // Geräte-ID (z.B. '12345')
	 I_iInstID				:INT 	:=	17;
	 I_sReceivedString		:STRING(255);	
	 I_bReset				:BOOL;
END_VAR
VAR_OUTPUT
	Q_lrRhd					:LREAL;
	Q_bStartupDone			:BOOL;
	Q_tUpdate				:TIME;
	Q_sLastUpdate			:STRING(12);
END_VAR
VAR	
	findStringTemp			:STRING(255);	(* Wird für TMP/ BRS/ RHD verwendet *)

	sTemp1					:STRING(255);
	sTemp2					:STRING(255);
	
	startPos : INT;
		
	iFindString	:int;
	icnt					:INT ;
	r_trigCnt				:r_trig;
	
	bStartupStart			:BOOL;
	bStartupDone			:BOOL;
	
	iStartup				:INT;	
	
	fbtimeDiff				:fb_timeDiffLite_libversion;
	bUpdated				: BOOL;
	
	sLastString				:STRING(255);
	bNeedProcess			:BOOL;
END_VAR

r_trigCnt();

(* Automatische Fehlererkennung *)
IF NOT I_bExecute
	OR (I_diID = 0)
	OR (I_iInstID = 0)
THEN
	iStartup := 0;
END_IF

(* Warten, ob der String sich geändert hat*)
bNeedProcess :=	(I_sReceivedString <> sLastString) 
				AND (I_sReceivedString <> '');
				
CASE iStartup OF 
(*=====================================*)
0 :	(* INIT *)
	bStartupDone := FALSE;
	bStartupStart := FALSE;
	sTemp2 :=sTemp1 := '0';
	r_trigCnt.CLK := FALSE;
	bNeedProcess := FALSE;
	sLastString := '';
	
	IF I_bExecute
		AND NOT bStartupDone
		AND NOT I_bReset
		AND (I_diID <> 0)
		AND (I_iInstID <>0)
	THEN
		bStartupStart := TRUE;
		iStartup := iStartup +10;
	END_IF
	
(*=====================================*)
10 :(* String vorbereiten *)	
	
	findStringTemp := F_RS485HB_TO_ASCII_RX(
								I_diID			:= I_diID, 
								I_iInstID		:= I_iInstID,	
								I_EnumHBUnitTX	:= E_EnumHBUnitTX.E_HB_UNIT_RHD, 	
								I_EnumHBCmdRX	:= E_EnumHBCmdRX.E_HB_CMD_STATUS , 
								I_iP1			:= 0);
	iStartup := 999;
	
(*=====================================*)
999 :(* READY *)
	bStartupDone := TRUE;
	
	IF I_bReset 
	THEN
		iStartup := 0;
	ELSE
		IF bNeedProcess
		THEN
			iFindString :=	FIND(I_sReceivedString,findStringTemp);
			
			IF iFindString>0
			THEN
				r_trigCnt.CLK := TRUE;
				startPos := iFindString; // Position des Suchstrings       
				(*Temperatur steht direkt nach dem Suchstring*)
				startPos := startPos + LEN(findStringTemp); (*Startposition für Temperatur*)
				(* Temperatur bis zum nächsten Komma oder Ende auslesen (maximal 6 Zeichen: z.B. 24,74)*)
				sTemp1 := MID(I_sReceivedString, 5, startPos);
				(*Dezimalpunkt für STRING_TO_LREAL anpassen, falls nötig *)
				sTemp1 := REPLACE(sTemp1, '.',1,3); (* 1. Vorkommen ersetzen *)
			ELSE
				r_trigCnt.CLK := FALSE;
			END_IF
			
			sLastString :=	I_sReceivedString;	(* Letzten String Speichern *)
		END_IF
	END_IF
		
	
	Q_lrRhd := STRING_TO_LREAL(sTemp1);
	
	(* Counter für Diagnose *)
	IF r_trigCnt.Q
	THEN
		Q_sLastUpdate :=	sGlobClock_SMH;	(* Globale Uhrzeit SMH*)
		
		bUpdated := TRUE;
		sTemp2 :=	I_sReceivedString;	(* Speichern der Werte *)
		icnt := icnt+1;
	ELSE
		bUpdated := FALSE;
	END_IF
	
END_CASE

Q_bStartupDone := bStartupDone;

(*=====================================*)
(* Zeitmessung zwischen den Updates *)
fbtimeDiff(
	I_bStart:= 			bUpdated, 
	I_bReset:= 			I_bReset, 
	Q_tDiffTime=>		Q_tUpdate);

END_FUNCTION_BLOCK

// ---- POUs/RS485_Hausbus_FB/00_Events/fb_BusTasterAdvancedEvent_4F.TcPOU
(*======================================================================================================================================*)
(*//=============================================================================\\
||  _   _ _  __  _         _                        _   _                      ||
|| | \ | | |/ / / \  _   _| |_ ___  _ __ ___   __ _| |_(_) ___  _ __         ||
|| |  \| | ' / / _ \| | | | __/ _ \| '_ ` _ \ / _` | __| |/ _ \| '_ \        ||
|| | |\  | . \/ ___ \ |_| | || (_) | | | | | | (_| | |_| | (_) | | | |       ||
|| |_| \_|_|\_\_/  \_\__,_|\__\___/|_| |_| |_|\__,_|\__|_|\___/|_| |_|       ||
||                                                                             ||
\\=============================================================================//
fb_BusTasterAdvancedEvent:	Dieser Baustein sieht Taster Events und wertet diese aus, möglichst effizient.
								Die Vorgängerversion: fb_BusTasterEvent hat durchgehend die CONCAT funktion für die Erstellung der Suchstrings 
								genutzt, wodurch die CPU Last erhöht wurde.   *)
(*
Date          	| Version    	| created under        	| Author          	| Remark *)
(*====================================================================================================================================================*)
(*29/04/2025   	| 1.00      		| TC3		  		| N.Kersting       | first release *)
(*13/08/2025   	| 1.01      		| TC3		  		| N.Kersting       | Neuer Aufbau, um Leistung zu sparen wegen hoher CPU Auslastung *)
(*27/08/2025   	| 1.02      		| TC3		  		| N.Kersting       | Reset hinzugefügt *)
(*07/09/2025   	| 1.03      		| TC3		  		| N.Kersting       | Zykluszeit Optimierung, es wird nur gelesen, wenn String gefüllt ist *)
(*09/09/2025   	| 1.04      		| TC3		  		| N.Kersting       | Zykluszeit Optimierung, Wirklich nur einen Zyklus suchen *)
(*23/01/2026   	| 1.05      		| TC3		  		| N.Kersting       | Suchstring wird nun einheitlich mit der funktion: F_RS485HB_TO_ASCII_RX gebildet *)
(*25/01/2026   	| 2.00      		| TC3		  		| N.Kersting       | Suchstring umstellung auf ASCII_RS485 Funktion *)
(*26/01/2026   	| 2.01      		| TC3		  		| N.Kersting       | Erweiterung auf Angeforderte Suchstrings (rStatus) *)
(*====================================================================================================================================================*)
FUNCTION_BLOCK fb_BusTasterAdvancedEvent_4F
VAR_INPUT
	 I_bExecute				:BOOL := TRUE;	// Aktiviert den Baustein 
	 I_bReset				:BOOL;
	 I_diID         		:DINT;     // Geräte-ID (z.B. '12345')
	 I_iInstID				:INT 	:=	17;
	 I_sReceivedString		:STRING(255);	
	 I_bFaultDetection		:BOOL := FALSE;		(* Soll erkennen, ob ein Telegramm für das zurücksetzen eines Tasters nicht gekommen ist *)
	 I_tFaultDetectTime		:TIME := T#10S;
END_VAR
VAR_OUTPUT
	Q_bOut					:ARRAY[1..4] OF  BOOL;
	Q_bStartupDone			:BOOL;
END_VAR
VAR
	i						:INT;
	tonFaultInput			:ARRAY[1..4] OF ton;
	findString0				:ARRAY[1..4] OF STRING(255) ;
	findString1				:ARRAY[1..4] OF STRING(255) ;
	findString2				:ARRAY[1..4] OF STRING(255) ; 	(* Angeforderter Status AUS*)
	findString3				:ARRAY[1..4] OF STRING(255) ;	(* Angeforderter Status EIN *)
	
	bStartupStart			:BOOL;
	bStartupDone			:BOOL;
	
	iStartup				:INT;
	sLastString				:STRING(255);
	bNeedProcess			:BOOL;
END_VAR

(* Automatische Fehlererkennung *)
IF NOT I_bExecute
	OR (I_diID = 0)
	OR (I_iInstID = 0)
THEN
	iStartup := 0;
END_IF

(* Warten, ob der String sich geändert hat*)
bNeedProcess :=	(I_sReceivedString <> sLastString) 
				AND (I_sReceivedString <> '');

CASE iStartup OF 
(*=====================================*)
0 :	(* INIT *)
	bStartupDone := FALSE;
	bStartupStart := FALSE;
	bNeedProcess := FALSE;
	sLastString := '';
	
	FOR i := 1 TO 4 BY 1 DO
		
		Q_bOut[i] := FALSE;
		
		tonFaultInput[i](
			IN := FALSE);
	END_FOR	
	
	IF I_bExecute
		AND NOT bStartupDone
		AND NOT I_bReset
		AND (I_diID <> 0)
		AND (I_iInstID <>0)
	THEN
		i := 1;
		bStartupStart := TRUE;
		iStartup := iStartup +10;
	END_IF
	
(*=====================================*)
10 :(* String vorbereiten *)	
	
	FOR i := 1 TO 4 BY 1 DO
		findString0[i] := F_RS485HB_TO_ASCII_RX(
								I_diID			:= I_diID, 
								I_iInstID		:= I_iInstID+i,	
								I_EnumHBUnitTX	:= E_EnumHBUnitTX.E_HB_UNIT_BTN, 	
								I_EnumHBCmdRX	:= E_EnumHBCmdRX.E_HB_CMD_STATUS , 
								I_iP1			:= 0);
		
		findString1[i] := F_RS485HB_TO_ASCII_RX(
								I_diID			:= I_diID, 
								I_iInstID		:= I_iInstID+i,	
								I_EnumHBUnitTX	:= E_EnumHBUnitTX.E_HB_UNIT_BTN, 	
								I_EnumHBCmdRX	:= E_EnumHBCmdRX.E_HB_CMD_STATUS , 
								I_iP1			:= 1);
			
		findString2[i] := F_RS485HB_TO_ASCII_RX(
								I_diID			:= I_diID, 
								I_iInstID		:= I_iInstID+i,	
								I_EnumHBUnitTX	:= E_EnumHBUnitTX.E_HB_UNIT_BTN, 	
								I_EnumHBCmdRX	:= E_EnumHBCmdRX.E_HB_CMD_rSTATUS , 
								I_iP1			:= 0);
		
		findString3[i] := F_RS485HB_TO_ASCII_RX(
								I_diID			:= I_diID, 
								I_iInstID		:= I_iInstID+i,	
								I_EnumHBUnitTX	:= E_EnumHBUnitTX.E_HB_UNIT_BTN, 	
								I_EnumHBCmdRX	:= E_EnumHBCmdRX.E_HB_CMD_rSTATUS , 
								I_iP1			:= 1);
	END_FOR
	
	IF i >= 4 THEN
		bStartupStart := FALSE;
		iStartup := 999;
	END_IF
	
(*=====================================*)
999 :(* READY *)
	bStartupDone := TRUE;
	
	IF I_bReset 
	THEN
		iStartup := 0;
	ELSE
		IF bNeedProcess
		THEN
			FOR i := 1 TO 4 BY 1 DO			
				IF I_bFaultDetection
				THEN
					tonFaultInput[i](
						IN := Q_bOut[i],
						PT := I_tFaultDetectTime);
				END_IF
		
				IF ((FIND(I_sReceivedString,findString0[i]) <>0	(* Automatischer Status AUS*)
					OR FIND(I_sReceivedString,findString2[i]) <>0)  (* Angeforderter Status AUS*)
					AND Q_bOut[i])
					OR ( tonFaultInput[i].Q
						AND I_bFaultDetection)
				THEN
					Q_bOut[i] := FALSE;
				ELSIF
					((FIND(I_sReceivedString,findString1[i]) <>0 (* Automatischer Status EIN *)
						OR FIND(I_sReceivedString,findString3[i]) <>0)	(* Angeforderter Status EIN*)
					AND NOT Q_bOut[i])
				THEN
					Q_bOut[i] := TRUE;
				END_IF
			END_FOR
				
			sLastString :=	I_sReceivedString;	(* Letzten String Speichern *)
		END_IF
	END_IF
	
END_CASE

Q_bStartupDone := bStartupDone;

END_FUNCTION_BLOCK

// ---- POUs/RS485_Hausbus_FB/00_Events/fb_BusTasterAdvancedEvent_6F.TcPOU
(*======================================================================================================================================*)
(*//=============================================================================\\
||  _   _ _  __  _         _                        _   _                      ||
|| | \ | | |/ / / \  _   _| |_ ___  _ __ ___   __ _| |_(_) ___  _ __         ||
|| |  \| | ' / / _ \| | | | __/ _ \| '_ ` _ \ / _` | __| |/ _ \| '_ \        ||
|| | |\  | . \/ ___ \ |_| | || (_) | | | | | | (_| | |_| | (_) | | | |       ||
|| |_| \_|_|\_\_/  \_\__,_|\__\___/|_| |_| |_|\__,_|\__|_|\___/|_| |_|       ||
||                                                                             ||
\\=============================================================================//
fb_BusTasterAdvancedEvent:	Dieser Baustein sieht Taster Events und wertet diese aus, möglichst effizient.
								Die Vorgängerversion: fb_BusTasterEvent hat durchgehend die CONCAT funktion für die Erstellung der Suchstrings 
								genutzt, wodurch die CPU Last erhöht wurde.   *)
(*
Date          	| Version    	| created under        	| Author          	| Remark *)
(*====================================================================================================================================================*)
(*29/04/2025   	| 1.00      		| TC3		  		| N.Kersting       | first release *)
(*13/08/2025   	| 1.01      		| TC3		  		| N.Kersting       | Neuer Aufbau, um Leistung zu sparen wegen hoher CPU Auslastung *)
(*27/08/2025   	| 1.02      		| TC3		  		| N.Kersting       | Reset hinzugefügt *)
(*07/09/2025   	| 1.03      		| TC3		  		| N.Kersting       | Zykluszeit Optimierung, es wird nur gelesen, wenn String gefüllt ist *)
(*09/09/2025   	| 1.04      		| TC3		  		| N.Kersting       | Zykluszeit Optimierung, Wirklich nur einen Zyklus suchen *)
(*23/01/2026   	| 1.05      		| TC3		  		| N.Kersting       | Suchstring wird nun einheitlich mit der funktion: F_RS485HB_TO_ASCII_RX gebildet *)
(*25/01/2026   	| 2.00      		| TC3		  		| N.Kersting       | Suchstring umstellung auf ASCII_RS485 Funktion *)
(*26/01/2026   	| 2.01      		| TC3		  		| N.Kersting       | Erweiterung auf Angeforderte Suchstrings (rStatus) *)
(*====================================================================================================================================================*)
FUNCTION_BLOCK fb_BusTasterAdvancedEvent_6F
VAR_INPUT
	 I_bExecute				:BOOL := TRUE;	// Aktiviert den Baustein 
	 I_bReset				:BOOL;
	 I_diID         		:DINT;     // Geräte-ID (z.B. '12345')
	 I_iInstID				:INT 	:=	17;
	 I_sReceivedString		:STRING(255);	
	 I_bFaultDetection		:BOOL := FALSE;		(* Soll erkennen, ob ein Telegramm für das zurücksetzen eines Tasters nicht gekommen ist *)
	 I_tFaultDetectTime		:TIME := T#10S;
END_VAR
VAR_OUTPUT
	Q_bOut					:ARRAY[1..6] OF  BOOL;
	Q_bStartupDone			:BOOL;
END_VAR
VAR
	i						:INT;
	tonFaultInput			:ARRAY[1..6] OF ton;
	findString0				:ARRAY[1..6] OF STRING(255) ; 	(* Automatischer Status AUS*)
	findString1				:ARRAY[1..6] OF STRING(255) ;	(* Automatischer Status EIN *)
	findString2				:ARRAY[1..6] OF STRING(255) ; 	(* Angeforderter Status AUS*)
	findString3				:ARRAY[1..6] OF STRING(255) ;	(* Angeforderter Status EIN *)
	
	bStartupStart			:BOOL;
	bStartupDone			:BOOL;
	
	iStartup				:INT;
	sLastString				:STRING(255);
	bNeedProcess			:BOOL;
END_VAR

(* Automatische Fehlererkennung *)
IF NOT I_bExecute
	OR (I_diID = 0)
	OR (I_iInstID = 0)
THEN
	iStartup := 0;
END_IF

(* Warten, ob der String sich geändert hat*)
bNeedProcess :=	(I_sReceivedString <> sLastString) 
				AND (I_sReceivedString <> '');

CASE iStartup OF 
(*=====================================*)
0 :	(* INIT *)
	bStartupDone := FALSE;
	bStartupStart := FALSE;
	bNeedProcess := FALSE;
	sLastString := '';
	
	FOR i := 1 TO 6 BY 1 DO
		
		Q_bOut[i] := FALSE;
		
		tonFaultInput[i](
			IN := FALSE);
	END_FOR	
	
	IF I_bExecute
		AND NOT bStartupDone
		AND NOT I_bReset
		AND (I_diID <> 0)
		AND (I_iInstID <>0)
	THEN
		i := 1;
		bStartupStart := TRUE;
		iStartup := iStartup +10;
	END_IF
	
(*=====================================*)
10 :(* String vorbereiten *)	
	
	FOR i := 1 TO 6 BY 1 DO
		findString0[i] := F_RS485HB_TO_ASCII_RX(
								I_diID			:= I_diID, 
								I_iInstID		:= I_iInstID+i,	
								I_EnumHBUnitTX	:= E_EnumHBUnitTX.E_HB_UNIT_BTN, 	
								I_EnumHBCmdRX	:= E_EnumHBCmdRX.E_HB_CMD_STATUS , 
								I_iP1			:= 0);
		
		findString1[i] := F_RS485HB_TO_ASCII_RX(
								I_diID			:= I_diID, 
								I_iInstID		:= I_iInstID+i,	
								I_EnumHBUnitTX	:= E_EnumHBUnitTX.E_HB_UNIT_BTN, 	
								I_EnumHBCmdRX	:= E_EnumHBCmdRX.E_HB_CMD_STATUS , 
								I_iP1			:= 1);
				
		findString2[i] := F_RS485HB_TO_ASCII_RX(
								I_diID			:= I_diID, 
								I_iInstID		:= I_iInstID+i,	
								I_EnumHBUnitTX	:= E_EnumHBUnitTX.E_HB_UNIT_BTN, 	
								I_EnumHBCmdRX	:= E_EnumHBCmdRX.E_HB_CMD_rSTATUS , 
								I_iP1			:= 0);
		
		findString3[i] := F_RS485HB_TO_ASCII_RX(
								I_diID			:= I_diID, 
								I_iInstID		:= I_iInstID+i,	
								I_EnumHBUnitTX	:= E_EnumHBUnitTX.E_HB_UNIT_BTN, 	
								I_EnumHBCmdRX	:= E_EnumHBCmdRX.E_HB_CMD_rSTATUS , 
								I_iP1			:= 1);
	END_FOR
	
	IF i >= 6 THEN
		bStartupStart := FALSE;
		iStartup := 999;
	END_IF
	
(*=====================================*)
999 :(* READY *)
	bStartupDone := TRUE;
	
	IF I_bReset 
	THEN
		iStartup := 0;
	ELSE
		IF bNeedProcess
		THEN
			FOR i := 1 TO 6 BY 1 DO			
				IF I_bFaultDetection
				THEN
					tonFaultInput[i](
						IN := Q_bOut[i],
						PT := I_tFaultDetectTime);
				END_IF
		
				IF ((FIND(I_sReceivedString,findString0[i]) <>0	(* Automatischer Status AUS*)
					OR FIND(I_sReceivedString,findString2[i]) <>0)  (* Angeforderter Status AUS*)
					AND Q_bOut[i])
					OR ( tonFaultInput[i].Q
						AND I_bFaultDetection)
				THEN
					Q_bOut[i] := FALSE;
				ELSIF
					((FIND(I_sReceivedString,findString1[i]) <>0 (* Automatischer Status EIN *)
						OR FIND(I_sReceivedString,findString3[i]) <>0)	(* Angeforderter Status EIN*)
					AND NOT Q_bOut[i])
				THEN
					Q_bOut[i] := TRUE;
				END_IF
			END_FOR
				
			sLastString :=	I_sReceivedString;	(* Letzten String Speichern *)
		END_IF
	END_IF
	
END_CASE

Q_bStartupDone := bStartupDone;

END_FUNCTION_BLOCK

// ---- POUs/RS485_Hausbus_FB/00_Events/fb_BusTasterAdvancedEvent_8F.TcPOU
(*======================================================================================================================================*)
(*//=============================================================================\\
||  _   _ _  __  _         _                        _   _                      ||
|| | \ | | |/ / / \  _   _| |_ ___  _ __ ___   __ _| |_(_) ___  _ __         ||
|| |  \| | ' / / _ \| | | | __/ _ \| '_ ` _ \ / _` | __| |/ _ \| '_ \        ||
|| | |\  | . \/ ___ \ |_| | || (_) | | | | | | (_| | |_| | (_) | | | |       ||
|| |_| \_|_|\_\_/  \_\__,_|\__\___/|_| |_| |_|\__,_|\__|_|\___/|_| |_|       ||
||                                                                             ||
\\=============================================================================//
fb_BusTasterAdvancedEvent:	Dieser Baustein sieht Taster Events und wertet diese aus, möglichst effizient.
								Die Vorgängerversion: fb_BusTasterEvent hat durchgehend die CONCAT funktion für die Erstellung der Suchstrings 
								genutzt, wodurch die CPU Last erhöht wurde.   *)
(*
Date          	| Version    	| created under        	| Author          	| Remark *)
(*====================================================================================================================================================*)
(*29/04/2025   	| 1.00      		| TC3		  		| N.Kersting       | first release *)
(*13/08/2025   	| 1.01      		| TC3		  		| N.Kersting       | Neuer Aufbau, um Leistung zu sparen wegen hoher CPU Auslastung *)
(*27/08/2025   	| 1.02      		| TC3		  		| N.Kersting       | Reset hinzugefügt *)
(*07/09/2025   	| 1.03      		| TC3		  		| N.Kersting       | Zykluszeit Optimierung, es wird nur gelesen, wenn String gefüllt ist *)
(*09/09/2025   	| 1.04      		| TC3		  		| N.Kersting       | Zykluszeit Optimierung, Wirklich nur einen Zyklus suchen *)
(*23/01/2026   	| 1.05      		| TC3		  		| N.Kersting       | Suchstring wird nun einheitlich mit der funktion: F_RS485HB_TO_ASCII_RX gebildet *)
(*25/01/2026   	| 2.00      		| TC3		  		| N.Kersting       | Suchstring umstellung auf ASCII_RS485 Funktion *)
(*26/01/2026   	| 2.01      		| TC3		  		| N.Kersting       | Erweiterung auf Angeforderte Suchstrings (rStatus) *)
(*====================================================================================================================================================*)
FUNCTION_BLOCK fb_BusTasterAdvancedEvent_8F
VAR_INPUT
	 I_bExecute				:BOOL := TRUE;	// Aktiviert den Baustein 
	 I_bReset				:BOOL;
	 I_diID         		:DINT;     // Geräte-ID (z.B. '12345')
	 I_iInstID				:INT 	:=	17;
	 I_sReceivedString		:STRING(255);	
	 I_bFaultDetection		:BOOL := FALSE;		(* Soll erkennen, ob ein Telegramm für das zurücksetzen eines Tasters nicht gekommen ist *)
	 I_tFaultDetectTime		:TIME := T#10S;
END_VAR
VAR_OUTPUT
	Q_bOut					:ARRAY[1..8] OF  BOOL;
	Q_bStartupDone			:BOOL;
END_VAR
VAR
	i						:INT;
	tonFaultInput			:ARRAY[1..8] OF ton;
	findString0				:ARRAY[1..8] OF STRING(255) ;
	findString1				:ARRAY[1..8] OF STRING(255) ;
	findString2				:ARRAY[1..8] OF STRING(255) ; 	(* Angeforderter Status AUS*)
	findString3				:ARRAY[1..8] OF STRING(255) ;	(* Angeforderter Status EIN *)
	
	bStartupStart			:BOOL;
	bStartupDone			:BOOL;
	
	iStartup				:INT;
	sLastString				:STRING(255);
	bNeedProcess			:BOOL;
END_VAR

(* Automatische Fehlererkennung *)
IF NOT I_bExecute
	OR (I_diID = 0)
	OR (I_iInstID = 0)
THEN
	iStartup := 0;
END_IF

(* Warten, ob der String sich geändert hat*)
bNeedProcess :=	(I_sReceivedString <> sLastString) 
				AND (I_sReceivedString <> '');

CASE iStartup OF 
(*=====================================*)
0 :	(* INIT *)
	bStartupDone := FALSE;
	bStartupStart := FALSE;
	bNeedProcess := FALSE;
	sLastString := '';
	
	FOR i := 1 TO 8 BY 1 DO
		
		Q_bOut[i] := FALSE;
		
		tonFaultInput[i](
			IN := FALSE);
	END_FOR	
	
	IF I_bExecute
		AND NOT bStartupDone
		AND NOT I_bReset
		AND (I_diID <> 0)
		AND (I_iInstID <>0)
	THEN
		i := 1;
		bStartupStart := TRUE;
		iStartup := iStartup +10;
	END_IF
	
(*=====================================*)
10 :(* String vorbereiten *)	
	
	FOR i := 1 TO 8 BY 1 DO
		findString0[i] := F_RS485HB_TO_ASCII_RX(
								I_diID			:= I_diID, 
								I_iInstID		:= I_iInstID+i,	
								I_EnumHBUnitTX	:= E_EnumHBUnitTX.E_HB_UNIT_BTN, 	
								I_EnumHBCmdRX	:= E_EnumHBCmdRX.E_HB_CMD_STATUS , 
								I_iP1			:= 0);
		
		findString1[i] := F_RS485HB_TO_ASCII_RX(
								I_diID			:= I_diID, 
								I_iInstID		:= I_iInstID+i,	
								I_EnumHBUnitTX	:= E_EnumHBUnitTX.E_HB_UNIT_BTN, 	
								I_EnumHBCmdRX	:= E_EnumHBCmdRX.E_HB_CMD_STATUS , 
								I_iP1			:= 1);
								
		findString2[i] := F_RS485HB_TO_ASCII_RX(
								I_diID			:= I_diID, 
								I_iInstID		:= I_iInstID+i,	
								I_EnumHBUnitTX	:= E_EnumHBUnitTX.E_HB_UNIT_BTN, 	
								I_EnumHBCmdRX	:= E_EnumHBCmdRX.E_HB_CMD_rSTATUS , 
								I_iP1			:= 0);
		
		findString3[i] := F_RS485HB_TO_ASCII_RX(
								I_diID			:= I_diID, 
								I_iInstID		:= I_iInstID+i,	
								I_EnumHBUnitTX	:= E_EnumHBUnitTX.E_HB_UNIT_BTN, 	
								I_EnumHBCmdRX	:= E_EnumHBCmdRX.E_HB_CMD_rSTATUS , 
								I_iP1			:= 1);
	END_FOR
	
	IF i >= 8 THEN
		bStartupStart := FALSE;
		iStartup := 999;
	END_IF
	
(*=====================================*)
999 :(* READY *)
	bStartupDone := TRUE;
	
	IF I_bReset 
	THEN
		iStartup := 0;
	ELSE
		IF bNeedProcess
		THEN
			FOR i := 1 TO 8 BY 1 DO			
				IF I_bFaultDetection
				THEN
					tonFaultInput[i](
						IN := Q_bOut[i],
						PT := I_tFaultDetectTime);
				END_IF
		
				IF ((FIND(I_sReceivedString,findString0[i]) <>0	(* Automatischer Status AUS*)
					OR FIND(I_sReceivedString,findString2[i]) <>0)  (* Angeforderter Status AUS*)
					AND Q_bOut[i])
					OR ( tonFaultInput[i].Q
						AND I_bFaultDetection)
				THEN
					Q_bOut[i] := FALSE;
				ELSIF
					((FIND(I_sReceivedString,findString1[i]) <>0 (* Automatischer Status EIN *)
						OR FIND(I_sReceivedString,findString3[i]) <>0)	(* Angeforderter Status EIN*)
					AND NOT Q_bOut[i])
				THEN
					Q_bOut[i] := TRUE;
				END_IF
			END_FOR
				
			sLastString :=	I_sReceivedString;	(* Letzten String Speichern *)
		END_IF
	END_IF
	
END_CASE

Q_bStartupDone := bStartupDone;

END_FUNCTION_BLOCK

// ---- POUs/RS485_Hausbus_FB/00_Events/fb_BusTempEvent.TcPOU
(*======================================================================================================================================*)
(*//=============================================================================\\
||  _   _ _  __  _         _                        _   _                      ||
|| | \ | | |/ / / \  _   _| |_ ___  _ __ ___   __ _| |_(_) ___  _ __         ||
|| |  \| | ' / / _ \| | | | __/ _ \| '_ ` _ \ / _` | __| |/ _ \| '_ \        ||
|| | |\  | . \/ ___ \ |_| | || (_) | | | | | | (_| | |_| | (_) | | | |       ||
|| |_| \_|_|\_\_/  \_\__,_|\__\___/|_| |_| |_|\__,_|\__|_|\___/|_| |_|       ||
||                                                                             ||
\\=============================================================================//
fb_BusTempEvent:				Dieser Baustein sieht Temperatur Events.  *)
(*
Date          	| Version    	| created under        	| Author          	| Remark *)
(*====================================================================================================================================================*)
(*29/04/2025   	| 1.00      		| TC3		  		| N.Kersting       | first release *)
(*14/08/2025   	| 1.01      		| TC3		  		| N.Kersting       | Startup Schrittkette Implementiert um Effizienter zu werden*)
(*27/08/2025   	| 1.02      		| TC3		  		| N.Kersting       | Reset hinzugefügt / Startup Done Ausgang *)
(*03/09/2025   	| 1.03      		| TC3		  		| N.Kersting       | Wenn der Wert sich erneuert, wird die Zeit gemessen zwischen den Updates *)
(*04/09/2025   	| 1.04      		| TC3		  		| N.Kersting       | Reagieren nun auch auf Statusanfrage  *)
(*07/09/2025   	| 1.05      		| TC3		  		| N.Kersting       | Zykluszeit Optimierung, es wird nur gelesen, wenn String gefüllt ist *)
(*09/09/2025   	| 1.04      		| TC3		  		| N.Kersting       | Zykluszeit Optimierung, Wirklich nur einen Zyklus suchen *)
(*25/01/2026   	| 2.00      		| TC3		  		| N.Kersting       | Suchstring umstellung auf ASCII_RS485 Funktion *)
(*====================================================================================================================================================*)
FUNCTION_BLOCK fb_BusTempEvent
VAR_INPUT
	 I_bExecute				:BOOL := TRUE;	// Aktiviert den Baustein 
	 I_diID        			:DINT;     // Geräte-ID (z.B. '12345')
	 I_iInstID				:INT 	:=	17;
	 I_sReceivedString		:STRING(255);	
	 I_bReset				:BOOL;
END_VAR
VAR_OUTPUT
	Q_lrTemp				:LREAL;
	Q_bStartupDone			:BOOL;
	Q_tUpdate				:TIME;
	Q_sLastUpdate			:STRING(12);
END_VAR
VAR	
	findStringTemp			:STRING(255);	(* Wird für TMP/ BRS/ RHD verwendet *)
	findStringTemp1			:STRING(255);	(* Wird für TMP/ BRS/ RHD verwendet *)
	
	sTemp1					:STRING(255);
	sTemp2					:STRING(255);
	
	startPos 				: INT;
		
	iFindString				:INT;
	iFindString1			:INT;
	
	icnt					:INT ;
	r_trigCnt				:r_trig;
		
	bStartupStart			:BOOL;
	bStartupDone			:BOOL;
	
	iStartup				:INT;	
	fbtimeDiff				:fb_timeDiffLite_libversion;
	bUpdated				: BOOL;
	
	sLastString				:STRING(255);
	bNeedProcess			:BOOL;
END_VAR

r_trigCnt();

(* Automatische Fehlererkennung *)
IF NOT I_bExecute
	OR (I_diID = 0)
	OR (I_iInstID = 0)
THEN
	iStartup := 0;
END_IF

(* Warten, ob der String sich geändert hat*)
bNeedProcess :=	(I_sReceivedString <> sLastString) 
				AND (I_sReceivedString <> '');
				
CASE iStartup OF 
(*=====================================*)
0 :	(* INIT *)
	bStartupDone := FALSE;
	bStartupStart := FALSE;
	sTemp2 :=sTemp1 := '0';
	r_trigCnt.CLK := FALSE;
	bNeedProcess := FALSE;
	sLastString := '';
	
	IF I_bExecute
		AND NOT bStartupDone
		AND NOT I_bReset
		AND (I_diID <> 0)
		AND (I_iInstID <>0)
	THEN
		bStartupStart := TRUE;
		iStartup := iStartup +10;
	END_IF
	
(*=====================================*)
10 :(* String vorbereiten *)	
		
	findStringTemp := F_RS485HB_TO_ASCII_RX(
							I_diID			:= I_diID, 
							I_iInstID		:= I_iInstID,	
							I_EnumHBUnitTX	:= E_EnumHBUnitTX.E_HB_UNIT_TMP, 	
							I_EnumHBCmdRX	:= E_EnumHBCmdRX.E_HB_CMD_STATUS , 
							I_iP1			:= 0);
	
	findStringTemp1 := F_RS485HB_TO_ASCII_RX(
							I_diID			:= I_diID, 
							I_iInstID		:= I_iInstID,	
							I_EnumHBUnitTX	:= E_EnumHBUnitTX.E_HB_UNIT_TMP, 	
							I_EnumHBCmdRX	:= E_EnumHBCmdRX.E_HB_CMD_rSTATUS , 
							I_iP1			:= 0);
						
	iStartup := 999;
	
(*=====================================*)
999 :(* READY *)
		
	bStartupDone := TRUE;
	
	IF I_bReset 
	THEN
		iStartup :=0;
	ELSE
		IF bNeedProcess
		THEN
			iFindString :=	FIND(I_sReceivedString,findStringTemp);
			iFindString1 :=	FIND(I_sReceivedString,findStringTemp1);
			
			IF iFindString>0
				AND  iFindString1 =0
			THEN
				r_trigCnt.CLK := TRUE;
				startPos := iFindString; // Position des Suchstrings       
				(*Temperatur steht direkt nach dem Suchstring*)
				startPos := startPos + LEN(findStringTemp); (*Startposition für Temperatur*)
				(* Temperatur bis zum nächsten Komma oder Ende auslesen (maximal 6 Zeichen: z.B. 24,74)*)
				sTemp1 := MID(I_sReceivedString, 5, startPos);
				(*Dezimalpunkt für STRING_TO_LREAL anpassen, falls nötig *)
				sTemp1 := REPLACE(sTemp1, '.',1,3); (* 1. Vorkommen ersetzen *)
				
			ELSIF iFindString1>0	
			THEN
				(* Neu, damit auch bei Statusabfragen reagiert werden kann *)
				r_trigCnt.CLK := TRUE;
				startPos := iFindString1; // Position des Suchstrings       
				(*Temperatur steht direkt nach dem Suchstring*)
				startPos := startPos + LEN(findStringTemp1); (*Startposition für Temperatur*)
				(* Temperatur bis zum nächsten Komma oder Ende auslesen (maximal 6 Zeichen: z.B. 24,74)*)
				sTemp1 := MID(I_sReceivedString, 5, startPos);
				(*Dezimalpunkt für STRING_TO_LREAL anpassen, falls nötig *)
				sTemp1 := REPLACE(sTemp1, '.',1,3); (* 1. Vorkommen ersetzen *)
			ELSE
				r_trigCnt.CLK := FALSE;
			END_IF
			
			sLastString :=	I_sReceivedString;	(* Letzten String Speichern *)
		END_IF
	END_IF
		
	
	Q_lrTemp := STRING_TO_LREAL(sTemp1);
	
	(* Counter für Diagnose *)
	IF r_trigCnt.Q
	THEN
		Q_sLastUpdate :=	sGlobClock_SMH;	(* Globale Uhrzeit SMH*)
		
		bUpdated := TRUE;
		sTemp2 :=	I_sReceivedString;	(* Speichern der Werte *)
		icnt := icnt+1;
	ELSE
		bUpdated := FALSE;
	END_IF
		
END_CASE

Q_bStartupDone := bStartupDone;

(*=====================================*)
(* Zeitmessung zwischen den Updates *)
fbtimeDiff(
	I_bStart:= 			bUpdated, 
	I_bReset:= 			I_bReset, 
	Q_tDiffTime=>		Q_tUpdate);

END_FUNCTION_BLOCK

// ---- POUs/RS485_Hausbus_FB/00_RS485 COM/FB/fb_FilterArray.TcPOU
(*======================================================================================================================================*)
(* Dieser Baustein Filtert eine Lreal Variable durch bildung eines Mittelwerts
(*======================================================================================================================================*)						

Date          		| Version    		| created under        		| Author          		| Remark *)
(*======================================================================================================================================*)
(*´10/07/2024   	| 1.00      			| TC2			  		| N.Kersting       	| first release *)
(*´15/07/2024   	| 1.01      			| TC2			  		| N.Kersting       	| Filterung nun Variabel einstellbar *)
(*======================================================================================================================================*)
FUNCTION_BLOCK fb_FilterArray
VAR_INPUT
	I_bExcecute	:BOOL;
	I_nWert		:LREAL;
	I_nFilterWert	:INT	:= 10;
END_VAR
VAR_OUTPUT
	Q_nFilter		:LREAL;
END_VAR
VAR
	i	:INT;
	nWertArray	:ARRAY [0..50] OF LREAL;
END_VAR

IF I_bExcecute THEN
   (* // Verschieben der Werte im Array*)
    FOR i := I_nFilterWert - 1 TO 1 BY -1 DO
        nWertArray[i] := nWertArray[i - 1];
    END_FOR

   (* // Neuen Wert einfügen	*)
    nWertArray[0] := I_nWert;

  (*  // Berechnung des gefilterten Wertes*)
    Q_nFilter := 0;
    FOR i := 0 TO I_nFilterWert - 1 DO
        Q_nFilter := Q_nFilter + nWertArray[i];
    END_FOR
    Q_nFilter := Q_nFilter / I_nFilterWert;

ELSE
  (*  // Initialisieren des Arrays*)
    FOR i := 0 TO 10 DO
        nWertArray[i] := 0;
    END_FOR
    Q_nFilter := 0;
END_IF

// ---- POUs/RS485_Hausbus_FB/00_RS485 COM/fb_RS485IdScan.TcPOU
(*======================================================================================================================================*)
(*//=============================================================================\\
||  _   _ _  __  _         _                        _   _                      ||
|| | \ | | |/ / / \  _   _| |_ ___  _ __ ___   __ _| |_(_) ___  _ __         ||
|| |  \| | ' / / _ \| | | | __/ _ \| '_ ` _ \ / _` | __| |/ _ \| '_ \        ||
|| | |\  | . \/ ___ \ |_| | || (_) | | | | | | (_| | |_| | (_) | | | |       ||
|| |_| \_|_|\_\_/  \_\__,_|\__\___/|_| |_| |_|\__,_|\__|_|\___/|_| |_|       ||
||                                                                             ||
\\=============================================================================//
fb_RS485Search:	Suchfunktion um Automatisch alle ID's im Bus zu Scannen*)
(*
Date          	| Version    	| created under        	| Author          	| Remark *)
(*====================================================================================================================================================*)
(*03/06/2025   	| 1.00      		| TC3		  		| N.Kersting       | first release *)
(*====================================================================================================================================================*)
FUNCTION_BLOCK fb_RS485IdScan
VAR_INPUT
	I_bStartSearch		:BOOL;
	I_diStartID			:DINT	:= 5000;
	I_diMaxID			:DINT	:= 6000;
	I_sStartZeichen		:BYTE := 16#FD;										(* Startzeichen Präfix *)
	I_sEndZeichen		:BYTE := 16#FE;										(* Endzeichen Suffix *)
	I_tWait				:TIME := T#300MS;
	I_StringReceived	:STRING(255);
END_VAR
VAR_OUTPUT
	Q_bSend				:BOOL;
	Q_sSearchString		:STRING(255);
	Q_iCnt				:INT;
	Q_sState			:STRING;
	Q_sIDList			:ARRAY[1..cMaxScanIDs] OF DINT;
END_VAR
VAR
	i					:INT;
	iArrIdx				:INT := 1;
	fbPingEvent			:fb_BusPingEvent;
	diActId				:DINT;
	iStep				:INT;
	tonWait				:ton;
	rTrigSearch			:r_trig;
END_VAR


tonWait(
	PT := I_tWait);
	
rTrigSearch(CLK:= I_bStartSearch, Q=> );

IF NOT I_bStartSearch
THEN
	iStep := 0;
END_IF
	
CASE iStep OF
(*=========================================================================*)
0:	Q_sState := 'INIT';
	tonWait.IN := FALSE;
	Q_bSend := FALSE;
	diActId := I_diStartID;
	Q_sSearchString := '';
	iArrIdx := 1;
	Q_iCnt := 0;
	
	IF rTrigSearch.Q
		AND I_diStartID >0
		AND I_diMaxID >0
	THEN
		FOR i := 1 TO cMaxScanIDs BY 1 DO 
			Q_sIDList[i] := 0;
		END_FOR
		
		iStep := iStep +1;
	END_IF
	
(*=========================================================================*)
1:	Q_bSend := FALSE;
	tonWait.IN := FALSE;
	
	IF diActId <= I_diMaxID
	THEN		
		iStep := iStep +1;
	ELSE
		iStep := 0;
	END_IF
	
(*=========================================================================*)
2:	Q_sSearchString := CONCAT(F_ToCHR(I_sStartZeichen),DINT_TO_STRING(diActId));
	Q_sSearchString := CONCAT(Q_sSearchString,'.TMP.1.gSTATUS');
	Q_sSearchString := CONCAT(Q_sSearchString,F_ToCHR(I_sEndZeichen));
	Q_sSearchString := CONCAT(Q_sSearchString,F_ToCHR(I_sStartZeichen));
	Q_sSearchString := CONCAT(Q_sSearchString,DINT_TO_STRING(diActId));
	Q_sSearchString := CONCAT(Q_sSearchString,'.OUT.210.gSTATUS');
	Q_sSearchString := CONCAT(Q_sSearchString,F_ToCHR(I_sEndZeichen));
	
	iStep := iStep +1;
	
(*=========================================================================*)
3:	Q_sState := 'Suchen Aktiv';
	tonWait.IN := TRUE;
	Q_bSend := TRUE;
	
	fbPingEvent(
		I_diID:= 				diActId, 
		I_sReceivedString:= 	I_StringReceived, 
		I_bReset:= ,
		Q_bOut=> );
		
	IF fbPingEvent.Q_bOut
	THEN
		Q_bSend := FALSE;
		iStep := iStep +1;
	ELSIF
		tonWait.Q
	THEN
		Q_bSend := FALSE;
		IF diActId <I_diMaxID
		THEN
			diActId := diActId +1;
			iStep := 1; (* nächsten Teilnehmer Suchen *)
		ELSE
			iStep := 6;	(* Scan Fertig *)
		END_IF
	END_IF
	
(*=========================================================================*)
4:	(* Teilnehmer gefunden ! *)
	Q_sState := 'Teilnehmer gefunden!';
	tonWait.IN := FALSE;	
	Q_bSend := FALSE;
	Q_sIDList[iArrIdx] := diActId;
	
	IF diActId <I_diMaxID
	THEN
		IF iArrIdx < cMaxScanIDs 
		THEN
			diActId := diActId +1;
			iArrIdx := iArrIdx +1;
			iStep := 1; (* nächsten Teilnehmer Suchen *)
		ELSE
			iStep := 5;
		END_IF
	ELSE
		iStep := 6;	(* Scan Fertig *)
	END_IF
	
(*=========================================================================*)
5:	(* Liste Voll! *)
	Q_sState := 'Liste Voll!';
	
(*=========================================================================*)
6:	(* Scan Fertig *)
	Q_iCnt := 0;
	
	FOR i := 1 TO cMaxScanIDs BY 1 DO 
		IF Q_sIDList[i] <> 0
		THEN
			Q_iCnt := Q_iCnt+1;
		END_IF
	END_FOR
	
	Q_sState := CONCAT('Scan Fertig! Es wurden: ',INT_TO_STRING(Q_iCnt));
	Q_sState := CONCAT(Q_sState,' Teilnehmer gefunden!');
		
	IF rTrigSearch.Q
	THEN
		iStep := 0;
	END_IF
END_CASE

END_FUNCTION_BLOCK

// ---- POUs/RS485_Hausbus_FB/00_RS485 COM/OLD/fb_RS485Ping.TcPOU
(*======================================================================================================================================*)
(*fb_RS485Ping:	Einfacher Universal Ping Baustein um von allerlei Geräten von haus-bus.de Kommunikation zu Checken über RS485 
				im gegensatz zum ComCheck Baustein wird hier nur gelesen, da es Geräte gibt, welche entweder Zyklich selbst 
				ein Lebenszeichen geben z.B. CYD oder die 6Fach Taster (Helligkeit, Temp, Luftfeuchtigkeit).
				Besonderheit bei dem 6Fach Taster ist: nach einem Reset werden immer auch StatusTelegramme gesendet. 
				Damit lässt sich dann auch festellen ob ein Taster Online ist. 
				Für die Aktoren ist dieser Baustein eher weniger geeignet, da es dort keine Zyklischen Telegramme gibt und 
				auch nach einem Reset keine Statustelegramme gesendet werden! 
				
				Der Baustein kann auch verwendet werden um einfach nur zu überwachen, ob ein Teilnehmer noch online ist über langen
				Zeitraum- Dafür muss der Timeout einfach sehr Hoch gestellt werden - z.B 120 Minuten und bAutoPing Aktiviert sein 
			
				Wenn I_bAutoPing nicht Aktiv ist, wird nur eine Ping überprüfung beim Aktivieren des Bausteins über I_bExecute 
				durchgeführt. Wenn die Prüfung erfolgreich ist, wird der Status Q_bComOk gesetzt. Der Status Q_bComOk wird erst durch 
				I_bReset wieder zurück gesetzt. 
				
				Wenn I_bAutoPing Aktiv ist, wird sobald der Baustein über I_bExecute gestartet wurde, und ein Ping Aufgebaut ist, 
				immer nach ablauf der Zeit: I_tPingTimeout erneut der Ping geprüft. Sollte der Ping nicht kommen, so wird nach ablauf der 
+				Zeit: I_tPingTimeout in den Timepout gesprungen. Dann kann nur über einen Reset durch: I_bReset erneut gestartet werden*)
(*
Date          	| Version    	| created under        	| Author          	| Remark *)
(*====================================================================================================================================================*)
(*27/05/2025   	| 1.00      		| TC3		  		| N.Kersting       | first release *)
(*27/08/2025   	| 1.01      		| TC3		  		| N.Kersting       | Startup für Eventbaustein Implementiert *)
(*====================================================================================================================================================*)
FUNCTION_BLOCK fb_RS485Ping
VAR_INPUT
	I_bExecute			:BOOL;							(* Aktiviert den Ablauf *)
	I_bAutoPing			:BOOL;							(* Aktiviert die Automatische Prüfung, wenn aus- wird nur einmal beim Aktivieren über bExecute geprüft *)
	I_bAutoReset		:BOOL;							(* Aktiviert das Automatische wieder Quittieren wenn der Ping nicht empfangen wurde *)
	I_bReset			:BOOL;							(* Setzet den Ping und die Ablauf zurück *)
	I_tPingTimeout		:TIME := T#2S;					(* Zeit, bis der Ping gekommen sein muss *)
	I_diID				:DINT;							(* Device ID *)
	I_sStartZeichen		:BYTE := 16#FD;					(* Startzeichen Präfix *)
	I_sEndZeichen		:BYTE := 16#FE;					(* Endzeichen Suffix *)
	I_StringReceived	:STRING(255);					(* Empfangener String *)
END_VAR
VAR_OUTPUT		
	Q_sState			:STRING;						(* Status  *)
	Q_bComOk			:BOOL;							(* Verbindung Aufgebaut *)
	Q_bTimeout			:BOOL;							(* Timeout  *)
END_VAR
VAR
	bResetCnt			:BOOL;
	tonTimeout			:ton;
	icntSymbole			:INT;
	iStep				:INT;
	i					:INT;
	fbBusPingEvent		:fb_BusPingEvent;
	bCOMMem				:BOOL;
	rTrigFailCount		:r_trig;
	
	dwCntFail			:DWORD;
	bResetEvents		:BOOL := FALSE;
END_VAR

(* Timeout Zeit *)
tonTimeout(
	PT:= I_tPingTimeout);

(* Ping Fehler Zählen *)	
rTrigFailCount();
	
(* Reset ausführen *)
IF I_bReset 
	OR NOT I_bExecute
THEN
	iStep := 0;	
END_IF

(* Timeout Counter auf 0 Setzen *)
IF bResetCnt
THEN
	dwCntFail := 0;
END_IF
	
(* Ablauf *)
CASE iStep OF
(*=========================================================*)	
0:	Q_sState := 'INIT';
	Q_bComOk := FALSE;
	bResetEvents := FALSE;	(*Alle Events Reset ausführen *)
	bCOMMem := FALSE; (* Ping zurück setzen *)
	tonTimeout.IN := FALSE;
	Q_bTimeout := FALSE;
	rTrigFailCount.CLK := FALSE;
	
	IF I_bExecute
	THEN
		iStep := iStep +1;
	END_IF

(*============================================================================================*)	
1:	Q_sState := 'Setze alle Eventbausteine zurück';
	
	bResetEvents := TRUE;	(*Alle Events Reset ausführen *)

	IF NOT fbBusPingEvent.Q_bStartupDone 
	THEN
		iStep := iStep +1;
	END_IF
	
(*============================================================================================*)	
2:	Q_sState := 'Warte auf Startup Eventbausteine';
	
	bResetEvents := FALSE;	(*Alle Events Reset ausführen *)

	IF  fbBusPingEvent.Q_bStartupDone 
	THEN
		iStep := 10;
	END_IF	
	
(*=========================================================*)	
10:	Q_sState :=  'Warten auf Ping ';	
	tonTimeout.IN := TRUE;
	
	IF fbBusPingEvent.Q_bOut
	THEN
		tonTimeout.IN := FALSE;
		bCOMMem := TRUE;
		iStep := 998;
	ELSIF
		tonTimeout.Q
	THEN
		tonTimeout.IN := FALSE;
		Q_bTimeout := TRUE;
		Q_bComOk := FALSE;
		Q_sState :=  'Timeout- Kein Ping empfangen';	
		iStep := -1;
	END_IF

(*=========================================================*)	
998: Q_sState :=  'Ping empfangen, Warte das String Leer ist';	
	tonTimeout.IN := TRUE;
	
	IF NOT fbBusPingEvent.Q_bOut
	THEN
		iStep := 999;
	ELSIF
		tonTimeout.Q
	THEN
		tonTimeout.IN := FALSE;
		Q_bTimeout := TRUE;
		Q_bComOk := FALSE;
		Q_sState :=  'Timeout String wurde nicht geleert!';	
		iStep := -998;
	END_IF
	
(*=========================================================*)	
999: Q_sState :=  'Ping empfangen, erfolgreich Verbunden!';		
	Q_bComOk := TRUE;
	Q_bTimeout := FALSE;
	
	(* Die Verbindung wurde nun geprüft, kann aber nur über
		I_bReset wieder erneut geprüft werden ! *)
	
	IF I_bAutoPing
	THEN
		tonTimeout.IN := TRUE;
		
		IF tonTimeout.Q
		THEN
			tonTimeout.IN := FALSE;
				
			IF I_bExecute
			THEN
				iStep := 10;	(* Erneut Prüfen *)
			END_IF
		END_IF
	ELSE
		tonTimeout.IN := FALSE;
	END_IF
ELSE
(*=========================================================*)	
(*	Timeout *)	
	rTrigFailCount.CLK := TRUE;
	
	IF rTrigFailCount.Q
	THEN
		dwCntFail := dwCntFail+1;
	END_IF
	(*	Automatische Quittierung *)	
	IF 	I_bAutoReset
	THEN
		tonTimeout.IN := TRUE;
		
		IF tonTimeout.Q
			OR fbBusPingEvent.Q_bOut
		THEN
			tonTimeout.IN := FALSE;
			
			IF I_bExecute
			THEN
				rTrigFailCount.CLK := FALSE;
				iStep := 10;	(* Erneut Prüfen *)
			END_IF
		END_IF
	END_IF
END_CASE

(* Durchgehend Checken ob Ping kommt *)
fbBusPingEvent(
	I_bExecute :=			TRUE,
	I_bReset := 			bResetEvents,
	I_diID:= 				I_diID, 
	I_sReceivedString:= 	I_StringReceived, 
	Q_bOut=> 				);

END_FUNCTION_BLOCK

// ---- POUs/RS485_Hausbus_FB/00_RS485 COM/RS485_Master/fb_RS485FiFoMaster.TcPOU
(*======================================================================================================================================*)
(*//=============================================================================\\
||  _   _ _  __  _         _                        _   _                      ||
|| | \ | | |/ / / \  _   _| |_ ___  _ __ ___   __ _| |_(_) ___  _ __         ||
|| |  \| | ' / / _ \| | | | __/ _ \| '_ ` _ \ / _` | __| |/ _ \| '_ \        ||
|| | |\  | . \/ ___ \ |_| | || (_) | | | | | | (_| | |_| | (_) | | | |       ||
|| |_| \_|_|\_\_/  \_\__,_|\__\___/|_| |_| |_|\__,_|\__|_|\___/|_| |_|       ||
||                                                                             ||
\\=============================================================================//
fb_RS485FiFoMaster:	Einfaches Senden eines Telegrams über RS485*)
(*
Date          	| Version    	| created under        	| Author          	| Remark *)
(*====================================================================================================================================================*)
(*10/05/2025   	| 1.00      		| TC3		  		| N.Kersting       | first release *)
(*10/05/2025   	| 1.01      		| TC3		  		| N.Kersting       | Nun wird der Empfang auch mit Implementiert  *)
(*13/05/2025   	| 1.02      		| TC3		  		| N.Kersting       | Busbelastungstest Implementiert - Sendet Durchgehend Strings *)
(*14/05/2025   	| 1.03      		| TC3		  		| N.Kersting       | Busauslastung direkt Implementiert *)
(*27/05/2025   	| 1.04      		| TC3		  		| N.Kersting       | Neuen Manuell Mode implementiert um einen Manuell generierten String allein zu Senden *)
(*28/05/2025   	| 1.05      		| TC3		  		| N.Kersting       | Neue Automatisch Ping Funktion hinzugefügt & Wichtiger Bugfix *)
(*02/06/2025   	| 2.00      		| TC3		  		| N.Kersting       | Neue Verbesserte Collision Detection, verhindert, dass Senden bei gefülltem Epmfangspuffer *)
(*03/06/2025   	| 2.01      		| TC3		  		| N.Kersting       | Collision Detection nun aufgeeilt in Empfang und Senden *)
(*03/06/2025   	| 2.02      		| TC3		  		| N.Kersting       | Neue Bus Scan Funktion Implementiert, Scannt alle Teilnehmer Ids im Bus (nur im Manuell Mode verfügbar) *)
(*12/01/2026   	| 2.03      		| TC3		  		| N.Kersting       | Nach dem Pingenkann wieder empfangen werden*)
(*13/01/2026   	| 2.04      		| TC3		  		| N.Kersting       | Ping wird Verzögert zwischen jedem Ping, wenn FiFo gefüllt kann Ping unterbrochen werden*)
(*13/01/2026   	| 2.04      		| TC3		  		| N.Kersting       | Bugfix Step 12 nur speichern wenn ID vorhanden ist!*)
(*09/06/2026   	| 2.05      		| TC3		  		| N.Kersting       | Obergrenze für Max Rows FiFo nun fix auf Globalen Wert *)
(*09/06/2026   	| 2.06      		| TC3		  		| N.Kersting       | Integration I_nMaxDevices*)
(*20/09/2026   	| 3.00      		| TC3		  		| N.Kersting       | Neue Parameter eingänge *)
(*====================================================================================================================================================*)
FUNCTION_BLOCK fb_RS485FiFoMaster
VAR_INPUT
	I_nMaxDevices				:INT := cMaxRowCMDFiFo;
	I_sSendCmdFiFo				:ARRAY[1..cMaxRowCMDFiFo] OF STRING(255);
	I_stDeviceIdent				:ARRAY[1..cMaxRowCMDFiFo] OF ST_HausBus_Ident;	(* Um Zyklisch einzelnt anzupingen *)
	
	I_bAutoPing					:BOOL;							(* Wenn Aktiv wird Zyklisch Automatisch ein Ping gesendet, welcher von den einzelnen Kommunikationsbausteinen ausgewertet werden kann *)
	I_tAutoPingTime				:TIME :=T#10S;					(* Die Intervallzeit, Bis ein Auto Ping gesendet wird *)
	
	I_bUseRXCollisionDetection	:BOOL := TRUE;					(* Aktiviert die Empfangs Kollisions Überprüfung -> Sollte immer an sein um Empfangstelegramme immer zu Proiorisieren!*)
	I_bUseTXCollisionDetection	:BOOL := FALSE;					(* Aktiviert die Sende Kollisions Überprüfung *)
	I_tVerzCollisionDetect		:TIME := T#100MS;				(* Collision detection Zeit *)
	I_tVerzPing					:TIME := T#100MS;				(* Verzögerung zischen denPings um sicher zu empfangen *)
	
	I_bManuellMode				:BOOL := FALSE;					(* Manueller Sendemodus *) 
	I_bSearchMode				:BOOL := FALSE;					(* Suchmodus Starten *)
	I_sSendCmdManuell			:STRING(255);					(* String, der beim Manuellen Modus gesendet wird *)
	I_bSendManuell				:BOOL := FALSE;					(* Manuelles Senden im Manuellen Sendemodus -> eigene Strings können eingegeben werden *)
	I_bLogger					:BOOL := FALSE;					(* Logger Starten *)
	I_bResetLog					:BOOL := FALSE;					(* Logger leeren *)
	I_bExecute					:BOOL := TRUE;					(* resertviert/ keine Funktion *)
	I_bBusBelastungstest		:BOOL := FALSE;					(* Startet den Busbelastungstest *)
	I_bReset					:BOOL := FALSE; 				(* Fehler zurücksetzen *)
	I_sStartZeichen				:BYTE := 16#FD;					(* Startzeichen Präfix *)
	I_sEndZeichen				:BYTE := 16#FE;					(* Endzeichen Suffix *)
	I_pTxBuffer					:POINTER TO ComBuffer; 			(* Zeiger auf TX-Buffer*)
	I_pRxBuffer   				:POINTER TO ComBuffer;  		(* Zeiger auf RX-Buffer*)
END_VAR
VAR_OUTPUT
	Q_bSendDoneFiFo				:ARRAY[1..cMaxRowCMDFiFo] OF BOOL; (*GVL_RS485FiFoSend.bSendDoneFiFo[iFiFoRow]*)
	Q_sReceiveString			:STRING(255);		
	Q_lrBusAuslastung			:LREAL;
	Q_bBusy						:BOOL;
	Q_bDone						:BOOL;
	Q_bError					:BOOL;
	Q_sState					:STRING;
	Q_stStates					:ST_FiFoMaster_State;
END_VAR
VAR
(*==========================================================================================================*)
(* Parameter *)
(*==========================================================================================================*)
	bActivateSend				:BOOL := TRUE;					(* Aktiviert das Senden von Nachrichten *)
	bActivateReceive			:BOOL := TRUE;					(* Aktiviert das Empfangen von Nachrichten *)
	
	bUseRXCollisionDetection	:BOOL := TRUE;					(* Aktiviert die Empfangs Kollisions Überprüfung *)
	bUseTXCollisionDetection	:BOOL := FALSE;					(* Aktiviert die Sende Kollisions Überprüfung *)
	tVerzCollisionDetect		:TIME := T#100MS;				(* Zeit, die zum Empfangen bleibt *)
	tVerzDoneTimeout			:TIME := T#2S;					(* Erkennung, ob ein Done hängen gebleiben ist *)
(*==========================================================================================================*)	
	bRXCollisionDetected		:BOOL;
	bTXCollisionDetected		:BOOL;
	bCollisionFree				:BOOL;	
(*==========================================================================================================*)		
	bFirstCycle					:BOOL := TRUE;
	bStringSend					:BOOL := FALSE;
	bBusBelastungstest			:BOOL := FALSE;
	bBusAuslastung				:BOOL := TRUE;
	bPingStart					:BOOL;
	bBusyMem					:BOOL;
	bFiFoDone					:BOOL; (* Merker, dass eventuell ein Done nicht Quittiert wurde *)
(*==========================================================================================================*)	
	sReceivedMEMString			:STRING(255);
	sReceivedString				:STRING(255);
	sStep						:STRING;
	sString						:STRING(255);
	sStringSend					:STRING(255);
(*==========================================================================================================*)		
	iStep						:INT;
	iStepReceive				:INT;
	iMaxBufferBlocking			:INT := 20;
	icntError					:INT;
	iFiFoRow					:INT := 1;
	iCntFiFoDone				:INT :=0;
	icntFiFo					:INT;
	i,h							:INT;
	iStepFiFo					:INT;
	iPingRow					:INT;
	dwCntTimeout				:DWORD := 0;
(*==========================================================================================================*)		

	tonCollisionFree			:ton;	
	tonTimeout					:ton;
	tonPingIntervall			:ton;
	tonPingVerz					:ton;
	tonSend						:ton;
	tonFiFoDoneTimeout			:ton;
(*==========================================================================================================*)		
	rTrigSendManuell			:r_Trig;
	rTrigSendSearchMode			:r_trig;
	fbSend     					:SendString255;
	fbReceive   				:ReceiveString255;
	
	fbBusAuslastung				:fb_FilterArray;
	
	fbRS485Search				:fb_RS485IdScan;
	
	fbRS485Logger				:fb_RS485Logger;
	
END_VAR

(*============================================================================================*)
(* Laufzeit fehler *)
tonTimeout(
	PT:=T#1S);

tonFiFoDoneTimeout(
	PT := tVerzDoneTimeout);
	
bUseRXCollisionDetection := 	I_bUseRXCollisionDetection;
bUseTXCollisionDetection :=		I_bUseTXCollisionDetection;
tVerzCollisionDetect :=			I_tVerzCollisionDetect;

